3187: L P[3187] 800cm/min CNT100 COORD PTH ;
:SR[23]=$SCR_GRP[1].$MCH_POS_X;
:SR[24]=$SCR_GRP[1].$MCH_POS_Y;
3188: L P[3188] 800cm/min CNT100 COORD PTH ;
:SR[23]=$SCR_GRP[1].$MCH_POS_X;
:SR[24]=$SCR_GRP[1].$MCH_POS_Y;
3189: L P[3189] 800cm/min CNT100 COORD PTH ;
:SR[23]=$SCR_GRP[1].$MCH_POS_X;
:SR[24]=$SCR_GRP[1].$MCH_POS_Y;
3190: L P[3190] 800cm/min CNT100 COORD PTH ;
:SR[23]=$SCR_GRP[1].$MCH_POS_X;
:SR[24]=$SCR_GRP[1].$MCH_POS_Y;
3191: L P[3191] 800cm/min CNT100 COORD PTH ;
:SR[23]=$SCR_GRP[1].$MCH_POS_X;
:SR[24]=$SCR_GRP[1].$MCH_POS_Y;
3192: L P[3192] 800cm/min CNT100 COORD PTH ;
:SR[23]=$SCR_GRP[1].$MCH_POS_X;
:SR[24]=$SCR_GRP[1].$MCH_POS_Y;
3193: L P[3193] 800cm/min CNT100 COORD PTH ;
:SR[23]=$SCR_GRP[1].$MCH_POS_X;
:SR[24]=$SCR_GRP[1].$MCH_POS_Y;
3194: L P[3194] 800cm/min CNT100 COORD PTH ;
:SR[23]=$SCR_GRP[1].$MCH_POS_X;
:SR[24]=$SCR_GRP[1].$MCH_POS_Y;
3195: L P[3195] 800cm/min CNT100 COORD PTH ;
:SR[23]=$SCR_GRP[1].$MCH_POS_X;
:SR[24]=$SCR_GRP[1].$MCH_POS_Y;
3196: L P[3196] 800cm/min CNT100 COORD PTH ;
:SR[23]=$SCR_GRP[1].$MCH_POS_X;
:SR[24]=$SCR_GRP[1].$MCH_POS_Y;
3197: L P[3197] 800cm/min CNT100 COORD PTH ;
:SR[23]=$SCR_GRP[1].$MCH_POS_X;
:SR[24]=$SCR_GRP[1].$MCH_POS_Y;
3198: L P[3198] 800cm/min CNT100 COORD PTH ;
:SR[23]=$SCR_GRP[1].$MCH_POS_X;
:SR[24]=$SCR_GRP[1].$MCH_POS_Y;
3199: L P[3199] 800cm/min CNT100 COORD PTH ;
:SR[23]=$SCR_GRP[1].$MCH_POS_X;
:SR[24]=$SCR_GRP[1].$MCH_POS_Y;
3200: L P[3200] 800cm/min CNT100 COORD PTH ;
:SR[23]=$SCR_GRP[1].$MCH_POS_X;
:SR[24]=$SCR_GRP[1].$MCH_POS_Y;
3201: L P[3201] 800cm/min CNT100 COORD PTH ;
:SR[23]=$SCR_GRP[1].$MCH_POS_X;
:SR[24]=$SCR_GRP[1].$MCH_POS_Y;
3202: L P[3202] 800cm/min CNT100 COORD PTH ;
:SR[23]=$SCR_GRP[1].$MCH_POS_X;
:SR[24]=$SCR_GRP[1].$MCH_POS_Y;
3203: L P[3203] 800cm/min CNT100 COORD PTH ;
:SR[23]=$SCR_GRP[1].$MCH_POS_X;
:SR[24]=$SCR_GRP[1].$MCH_POS_Y;
3204: L P[3204] 800cm/min CNT100 COORD PTH ;
:SR[23]=$SCR_GRP[1].$MCH_POS_X;
:SR[24]=$SCR_GRP[1].$MCH_POS_Y;
3205: L P[3205] 800cm/min CNT100 COORD PTH ;
:SR[23]=$SCR_GRP[1].$MCH_POS_X;
:SR[24]=$SCR_GRP[1].$MCH_POS_Y;
3206: L P[3206] 800cm/min CNT100 COORD PTH ;
:SR[23]=$SCR_GRP[1].$MCH_POS_X;
:SR[24]=$SCR_GRP[1].$MCH_POS_Y;
3207: L P[3207] 800cm/min CNT100 COORD PTH ;
:SR[23]=$SCR_GRP[1].$MCH_POS_X;
:SR[24]=$SCR_GRP[1].$MCH_POS_Y;
3208: L P[3208] 800cm/min CNT100 COORD PTH ;
:SR[23]=$SCR_GRP[1].$MCH_POS_X;
:SR[24]=$SCR_GRP[1].$MCH_POS_Y;
3209: L P[3209] 800cm/min CNT100 COORD PTH ;
:SR[23]=$SCR_GRP[1].$MCH_POS_X;
:SR[24]=$SCR_GRP[1].$MCH_POS_Y;
3210: L P[3210] 800cm/min CNT100 COORD PTH ;
:SR[23]=$SCR_GRP[1].$MCH_POS_X;
:SR[24]=$SCR_GRP[1].$MCH_POS_Y;
3211: L P[3211] 800cm/min CNT100 COORD PTH ;
:SR[23]=$SCR_GRP[1].$MCH_POS_X;
:SR[24]=$SCR_GRP[1].$MCH_POS_Y;
3212: L P[3212] 800cm/min CNT100 COORD PTH ;
:SR[23]=$SCR_GRP[1].$MCH_POS_X;
:SR[24]=$SCR_GRP[1].$MCH_POS_Y;
3213: L P[3213] 800cm/min CNT100 COORD PTH ;
:SR[23]=$SCR_GRP[1].$MCH_POS_X;
:SR[24]=$SCR_GRP[1].$MCH_POS_Y;
3214: L P[3214] 800cm/min CNT100 COORD PTH ;
:SR[23]=$SCR_GRP[1].$MCH_POS_X;
:SR[24]=$SCR_GRP[1].$MCH_POS_Y;
3215: L P[3215] 800cm/min CNT100 COORD PTH ;
:SR[23]=$SCR_GRP[1].$MCH_POS_X;
:SR[24]=$SCR_GRP[1].$MCH_POS_Y;
3216: L P[3216] 800cm/min CNT100 COORD PTH ;
:SR[23]=$SCR_GRP[1].$MCH_POS_X;
:SR[24]=$SCR_GRP[1].$MCH_POS_Y;
3217: L P[3217] 800cm/min CNT100 COORD PTH ;
:SR[23]=$SCR_GRP[1].$MCH_POS_X;
:SR[24]=$SCR_GRP[1].$MCH_POS_Y;
3218: L P[3218] 800cm/min CNT100 COORD PTH ;
:SR[23]=$SCR_GRP[1].$MCH_POS_X;
:SR[24]=$SCR_GRP[1].$MCH_POS_Y;
3219: L P[3219] 800cm/min CNT100 COORD PTH ;
:SR[23]=$SCR_GRP[1].$MCH_POS_X;
:SR[24]=$SCR_GRP[1].$MCH_POS_Y;
3220: L P[3220] 800cm/min CNT100 COORD PTH ;
:SR[23]=$SCR_GRP[1].$MCH_POS_X;
:SR[24]=$SCR_GRP[1].$MCH_POS_Y;
3221: L P[3221] 800cm/min CNT100 COORD PTH ;
:SR[23]=$SCR_GRP[1].$MCH_POS_X;
:SR[24]=$SCR_GRP[1].$MCH_POS_Y;
3222: L P[3222] 800cm/min CNT100 COORD PTH ;
:SR[23]=$SCR_GRP[1].$MCH_POS_X;
:SR[24]=$SCR_GRP[1].$MCH_POS_Y;
3223: L P[3223] 800cm/min CNT100 COORD PTH ;
:SR[23]=$SCR_GRP[1].$MCH_POS_X;
:SR[24]=$SCR_GRP[1].$MCH_POS_Y;
3224: L P[3224] 800cm/min CNT100 COORD PTH ;
:SR[23]=$SCR_GRP[1].$MCH_POS_X;
:SR[24]=$SCR_GRP[1].$MCH_POS_Y;
3225: L P[3225] 800cm/min CNT100 COORD PTH ;
:SR[23]=$SCR_GRP[1].$MCH_POS_X;
:SR[24]=$SCR_GRP[1].$MCH_POS_Y;
3226: L P[3226] 800cm/min CNT100 COORD PTH ;
:SR[23]=$SCR_GRP[1].$MCH_POS_X;
:SR[24]=$SCR_GRP[1].$MCH_POS_Y;
3227: L P[3227] 800cm/min CNT100 COORD PTH ;
:SR[23]=$SCR_GRP[1].$MCH_POS_X;
:SR[24]=$SCR_GRP[1].$MCH_POS_Y;
3228: L P[3228] 800cm/min CNT100 COORD PTH ;
:SR[23]=$SCR_GRP[1].$MCH_POS_X;
:SR[24]=$SCR_GRP[1].$MCH_POS_Y;
3229: L P[3229] 800cm/min CNT100 COORD PTH ;
:SR[23]=$SCR_GRP[1].$MCH_POS_X;
:SR[24]=$SCR_GRP[1].$MCH_POS_Y;
3230: L P[3230] 800cm/min CNT100 COORD PTH ;
:SR[23]=$SCR_GRP[1].$MCH_POS_X;
:SR[24]=$SCR_GRP[1].$MCH_POS_Y;
3231: L P[3231] 800cm/min CNT100 COORD PTH ;
:SR[23]=$SCR_GRP[1].$MCH_POS_X;
:SR[24]=$SCR_GRP[1].$MCH_POS_Y;
3232: L P[3232] 800cm/min CNT100 COORD PTH ;
:SR[23]=$SCR_GRP[1].$MCH_POS_X;
:SR[24]=$SCR_GRP[1].$MCH_POS_Y;
3233: L P[3233] 800cm/min CNT100 COORD PTH ;
:SR[23]=$SCR_GRP[1].$MCH_POS_X;
:SR[24]=$SCR_GRP[1].$MCH_POS_Y;
3234: L P[3234] 800cm/min CNT100 COORD PTH ;
:SR[23]=$SCR_GRP[1].$MCH_POS_X;
:SR[24]=$SCR_GRP[1].$MCH_POS_Y;
3235: L P[3235] 800cm/min CNT100 COORD PTH ;
:SR[23]=$SCR_GRP[1].$MCH_POS_X;
:SR[24]=$SCR_GRP[1].$MCH_POS_Y;
3236: L P[3236] 800cm/min CNT100 COORD PTH ;
:SR[23]=$SCR_GRP[1].$MCH_POS_X;
:SR[24]=$SCR_GRP[1].$MCH_POS_Y;
3237: L P[3237] 800cm/min CNT100 COORD PTH ;
:SR[23]=$SCR_GRP[1].$MCH_POS_X;
:SR[24]=$SCR_GRP[1].$MCH_POS_Y;
3238: L P[3238] 800cm/min CNT100 COORD PTH ;
:SR[23]=$SCR_GRP[1].$MCH_POS_X;
:SR[24]=$SCR_GRP[1].$MCH_POS_Y;
3239: L P[3239] 800cm/min CNT100 COORD PTH ;
:SR[23]=$SCR_GRP[1].$MCH_POS_X;
:SR[24]=$SCR_GRP[1].$MCH_POS_Y;
3240: L P[3240] 800cm/min CNT100 COORD PTH ;
:SR[23]=$SCR_GRP[1].$MCH_POS_X;
:SR[24]=$SCR_GRP[1].$MCH_POS_Y;
3241: L P[3241] 800cm/min CNT100 COORD PTH ;
:SR[23]=$SCR_GRP[1].$MCH_POS_X;
:SR[24]=$SCR_GRP[1].$MCH_POS_Y;
3242: L P[3242] 800cm/min CNT100 COORD PTH ;
:SR[23]=$SCR_GRP[1].$MCH_POS_X;
:SR[24]=$SCR_GRP[1].$MCH_POS_Y;
3243: L P[3243] 800cm/min CNT100 COORD PTH ;
:SR[23]=$SCR_GRP[1].$MCH_POS_X;
:SR[24]=$SCR_GRP[1].$MCH_POS_Y;
3244: L P[3244] 800cm/min CNT100 COORD PTH ;
:SR[23]=$SCR_GRP[1].$MCH_POS_X;
:SR[24]=$SCR_GRP[1].$MCH_POS_Y;
3245: L P[3245] 800cm/min CNT100 COORD PTH ;
:SR[23]=$SCR_GRP[1].$MCH_POS_X;
:SR[24]=$SCR_GRP[1].$MCH_POS_Y;
3246: L P[3246] 800cm/min CNT100 COORD PTH ;
:SR[23]=$SCR_GRP[1].$MCH_POS_X;
:SR[24]=$SCR_GRP[1].$MCH_POS_Y;
3247: L P[3247] 800cm/min CNT100 COORD PTH ;
:SR[23]=$SCR_GRP[1].$MCH_POS_X;
:SR[24]=$SCR_GRP[1].$MCH_POS_Y;
3248: L P[3248] 800cm/min CNT100 COORD PTH ;
:SR[23]=$SCR_GRP[1].$MCH_POS_X;
:SR[24]=$SCR_GRP[1].$MCH_POS_Y;
3249: L P[3249] 800cm/min CNT100 COORD PTH ;
:SR[23]=$SCR_GRP[1].$MCH_POS_X;
:SR[24]=$SCR_GRP[1].$MCH_POS_Y;
3250: L P[3250] 800cm/min CNT100 COORD PTH ;
:SR[23]=$SCR_GRP[1].$MCH_POS_X;
:SR[24]=$SCR_GRP[1].$MCH_POS_Y;
3251: L P[3251] 800cm/min CNT100 COORD PTH ;
:SR[23]=$SCR_GRP[1].$MCH_POS_X;
:SR[24]=$SCR_GRP[1].$MCH_POS_Y;
3252: L P[3252] 800cm/min CNT100 COORD PTH ;
:SR[23]=$SCR_GRP[1].$MCH_POS_X;
:SR[24]=$SCR_GRP[1].$MCH_POS_Y;
3253: L P[3253] 800cm/min CNT100 COORD PTH ;
:SR[23]=$SCR_GRP[1].$MCH_POS_X;
:SR[24]=$SCR_GRP[1].$MCH_POS_Y;
3254: L P[3254] 800cm/min CNT100 COORD PTH ;
:SR[23]=$SCR_GRP[1].$MCH_POS_X;
:SR[24]=$SCR_GRP[1].$MCH_POS_Y;
3255: L P[3255] 800cm/min CNT100 COORD PTH ;
:SR[23]=$SCR_GRP[1].$MCH_POS_X;
:SR[24]=$SCR_GRP[1].$MCH_POS_Y;
3256: L P[3256] 800cm/min CNT100 COORD PTH ;
:SR[23]=$SCR_GRP[1].$MCH_POS_X;
:SR[24]=$SCR_GRP[1].$MCH_POS_Y;
3257: L P[3257] 800cm/min CNT100 COORD PTH ;
:SR[23]=$SCR_GRP[1].$MCH_POS_X;
:SR[24]=$SCR_GRP[1].$MCH_POS_Y;
3258: L P[3258] 800cm/min CNT100 COORD PTH ;
:SR[23]=$SCR_GRP[1].$MCH_POS_X;
:SR[24]=$SCR_GRP[1].$MCH_POS_Y;
3259: L P[3259] 800cm/min CNT100 COORD PTH ;
:SR[23]=$SCR_GRP[1].$MCH_POS_X;
:SR[24]=$SCR_GRP[1].$MCH_POS_Y;
3260: L P[3260] 800cm/min CNT100 COORD PTH ;
:SR[23]=$SCR_GRP[1].$MCH_POS_X;
:SR[24]=$SCR_GRP[1].$MCH_POS_Y;
3261: L P[3261] 800cm/min CNT100 COORD PTH ;
:SR[23]=$SCR_GRP[1].$MCH_POS_X;
:SR[24]=$SCR_GRP[1].$MCH_POS_Y;
3262: L P[3262] 800cm/min CNT100 COORD PTH ;
:SR[23]=$SCR_GRP[1].$MCH_POS_X;
:SR[24]=$SCR_GRP[1].$MCH_POS_Y;
3263: L P[3263] 800cm/min CNT100 COORD PTH ;
:SR[23]=$SCR_GRP[1].$MCH_POS_X;
:SR[24]=$SCR_GRP[1].$MCH_POS_Y;
3264: L P[3264] 800cm/min CNT100 COORD PTH ;
:SR[23]=$SCR_GRP[1].$MCH_POS_X;
:SR[24]=$SCR_GRP[1].$MCH_POS_Y;
3265: L P[3265] 800cm/min CNT100 COORD PTH ;
:SR[23]=$SCR_GRP[1].$MCH_POS_X;
:SR[24]=$SCR_GRP[1].$MCH_POS_Y;
3266: L P[3266] 800cm/min CNT100 COORD PTH ;
:SR[23]=$SCR_GRP[1].$MCH_POS_X;
:SR[24]=$SCR_GRP[1].$MCH_POS_Y;
3267: L P[3267] 800cm/min CNT100 COORD PTH ;
:SR[23]=$SCR_GRP[1].$MCH_POS_X;
:SR[24]=$SCR_GRP[1].$MCH_POS_Y;
3268: L P[3268] 800cm/min CNT100 COORD PTH ;
:SR[23]=$SCR_GRP[1].$MCH_POS_X;
:SR[24]=$SCR_GRP[1].$MCH_POS_Y;
3269: L P[3269] 800cm/min CNT100 COORD PTH ;
:SR[23]=$SCR_GRP[1].$MCH_POS_X;
:SR[24]=$SCR_GRP[1].$MCH_POS_Y;
3270: L P[3270] 800cm/min CNT100 COORD PTH ;
:SR[23]=$SCR_GRP[1].$MCH_POS_X;
:SR[24]=$SCR_GRP[1].$MCH_POS_Y;
3271: L P[3271] 800cm/min CNT100 COORD PTH ;
:SR[23]=$SCR_GRP[1].$MCH_POS_X;
:SR[24]=$SCR_GRP[1].$MCH_POS_Y;
3272: L P[3272] 800cm/min CNT100 COORD PTH ;
:SR[23]=$SCR_GRP[1].$MCH_POS_X;
:SR[24]=$SCR_GRP[1].$MCH_POS_Y;
3273: L P[3273] 800cm/min CNT100 COORD PTH ;
:SR[23]=$SCR_GRP[1].$MCH_POS_X;
:SR[24]=$SCR_GRP[1].$MCH_POS_Y;
3274: L P[3274] 800cm/min CNT100 COORD PTH ;
:SR[23]=$SCR_GRP[1].$MCH_POS_X;
:SR[24]=$SCR_GRP[1].$MCH_POS_Y;
3275: L P[3275] 800cm/min CNT100 COORD PTH ;
:SR[23]=$SCR_GRP[1].$MCH_POS_X;
:SR[24]=$SCR_GRP[1].$MCH_POS_Y;
3276: L P[3276] 800cm/min CNT100 COORD ;
:SR[23]=$SCR_GRP[1].$MCH_POS_X;
:SR[24]=$SCR_GRP[1].$MCH_POS_Y;
3277: L P[3277] 800cm/min CNT100 COORD PTH ;
:SR[23]=$SCR_GRP[1].$MCH_POS_X;
:SR[24]=$SCR_GRP[1].$MCH_POS_Y;
3278: L P[3278] 800cm/min CNT100 COORD PTH ;
:SR[23]=$SCR_GRP[1].$MCH_POS_X;
:SR[24]=$SCR_GRP[1].$MCH_POS_Y;
3279: L P[3279] 800cm/min CNT100 COORD PTH ;
:SR[23]=$SCR_GRP[1].$MCH_POS_X;
:SR[24]=$SCR_GRP[1].$MCH_POS_Y;
3280: L P[3280] 800cm/min CNT100 COORD PTH ;
:SR[23]=$SCR_GRP[1].$MCH_POS_X;
:SR[24]=$SCR_GRP[1].$MCH_POS_Y;
3281: L P[3281] 800cm/min CNT100 COORD PTH ;
:SR[23]=$SCR_GRP[1].$MCH_POS_X;
:SR[24]=$SCR_GRP[1].$MCH_POS_Y;
3282: L P[3282] 800cm/min CNT100 COORD PTH ;
:SR[23]=$SCR_GRP[1].$MCH_POS_X;
:SR[24]=$SCR_GRP[1].$MCH_POS_Y;
3283: L P[3283] 800cm/min CNT100 COORD PTH ;
:SR[23]=$SCR_GRP[1].$MCH_POS_X;
:SR[24]=$SCR_GRP[1].$MCH_POS_Y;
3284: L P[3284] 800cm/min CNT100 COORD PTH ;
:SR[23]=$SCR_GRP[1].$MCH_POS_X;
:SR[24]=$SCR_GRP[1].$MCH_POS_Y;
3285: L P[3285] 800cm/min CNT100 COORD PTH ;
:SR[23]=$SCR_GRP[1].$MCH_POS_X;
:SR[24]=$SCR_GRP[1].$MCH_POS_Y;
3286: L P[3286] 800cm/min CNT100 COORD PTH ;
:SR[23]=$SCR_GRP[1].$MCH_POS_X;
:SR[24]=$SCR_GRP[1].$MCH_POS_Y;
3287: L P[3287] 800cm/min CNT100 COORD PTH ;
:SR[23]=$SCR_GRP[1].$MCH_POS_X;
:SR[24]=$SCR_GRP[1].$MCH_POS_Y;
3288: L P[3288] 800cm/min CNT100 COORD PTH ;
:SR[23]=$SCR_GRP[1].$MCH_POS_X;
:SR[24]=$SCR_GRP[1].$MCH_POS_Y;
3289: L P[3289] 800cm/min CNT100 COORD PTH ;
:SR[23]=$SCR_GRP[1].$MCH_POS_X;
:SR[24]=$SCR_GRP[1].$MCH_POS_Y;
3290: L P[3290] 800cm/min CNT100 COORD PTH ;
:SR[23]=$SCR_GRP[1].$MCH_POS_X;
:SR[24]=$SCR_GRP[1].$MCH_POS_Y;
3291: L P[3291] 800cm/min CNT100 COORD PTH ;
:SR[23]=$SCR_GRP[1].$MCH_POS_X;
:SR[24]=$SCR_GRP[1].$MCH_POS_Y;
3292: L P[3292] 800cm/min CNT100 COORD PTH ;
:SR[23]=$SCR_GRP[1].$MCH_POS_X;
:SR[24]=$SCR_GRP[1].$MCH_POS_Y;
3293: L P[3293] 800cm/min CNT100 COORD PTH ;
:SR[23]=$SCR_GRP[1].$MCH_POS_X;
:SR[24]=$SCR_GRP[1].$MCH_POS_Y;
3294: L P[3294] 800cm/min CNT100 COORD PTH ;
:SR[23]=$SCR_GRP[1].$MCH_POS_X;
:SR[24]=$SCR_GRP[1].$MCH_POS_Y;
3295: L P[3295] 800cm/min CNT100 COORD PTH ;
:SR[23]=$SCR_GRP[1].$MCH_POS_X;
:SR[24]=$SCR_GRP[1].$MCH_POS_Y;
3296: L P[3296] 800cm/min CNT100 COORD PTH ;
:SR[23]=$SCR_GRP[1].$MCH_POS_X;
:SR[24]=$SCR_GRP[1].$MCH_POS_Y;
3297: L P[3297] 800cm/min CNT100 COORD PTH ;
:SR[23]=$SCR_GRP[1].$MCH_POS_X;
:SR[24]=$SCR_GRP[1].$MCH_POS_Y;
3298: L P[3298] 800cm/min CNT100 COORD PTH ;
:SR[23]=$SCR_GRP[1].$MCH_POS_X;
:SR[24]=$SCR_GRP[1].$MCH_POS_Y;
3299: L P[3299] 800cm/min CNT100 COORD PTH ;
:SR[23]=$SCR_GRP[1].$MCH_POS_X;
:SR[24]=$SCR_GRP[1].$MCH_POS_Y;
3300: L P[3300] 800cm/min CNT100 COORD PTH ;
:SR[23]=$SCR_GRP[1].$MCH_POS_X;
:SR[24]=$SCR_GRP[1].$MCH_POS_Y;
3301: L P[3301] 800cm/min CNT100 COORD PTH ;
:SR[23]=$SCR_GRP[1].$MCH_POS_X;
:SR[24]=$SCR_GRP[1].$MCH_POS_Y;
3302: L P[3302] 800cm/min CNT100 COORD PTH ;
:SR[23]=$SCR_GRP[1].$MCH_POS_X;
:SR[24]=$SCR_GRP[1].$MCH_POS_Y;
3303: L P[3303] 800cm/min CNT100 COORD PTH ;
:SR[23]=$SCR_GRP[1].$MCH_POS_X;
:SR[24]=$SCR_GRP[1].$MCH_POS_Y;
3304: L P[3304] 800cm/min CNT100 COORD PTH ;
:SR[23]=$SCR_GRP[1].$MCH_POS_X;
:SR[24]=$SCR_GRP[1].$MCH_POS_Y;
3305: L P[3305] 800cm/min CNT100 COORD PTH ;
:SR[23]=$SCR_GRP[1].$MCH_POS_X;
:SR[24]=$SCR_GRP[1].$MCH_POS_Y;
3306: L P[3306] 800cm/min CNT100 COORD PTH ;
:SR[23]=$SCR_GRP[1].$MCH_POS_X;
:SR[24]=$SCR_GRP[1].$MCH_POS_Y;
3307: L P[3307] 800cm/min CNT100 COORD PTH ;
:SR[23]=$SCR_GRP[1].$MCH_POS_X;
:SR[24]=$SCR_GRP[1].$MCH_POS_Y;
3308: L P[3308] 800cm/min CNT100 COORD PTH ;
:SR[23]=$SCR_GRP[1].$MCH_POS_X;
:SR[24]=$SCR_GRP[1].$MCH_POS_Y;
3309: L P[3309] 800cm/min CNT100 COORD PTH ;
:SR[23]=$SCR_GRP[1].$MCH_POS_X;
:SR[24]=$SCR_GRP[1].$MCH_POS_Y;
3310: L P[3310] 800cm/min CNT100 COORD PTH ;
:SR[23]=$SCR_GRP[1].$MCH_POS_X;
:SR[24]=$SCR_GRP[1].$MCH_POS_Y;
3311: L P[3311] 800cm/min CNT100 COORD PTH ;
:SR[23]=$SCR_GRP[1].$MCH_POS_X;
:SR[24]=$SCR_GRP[1].$MCH_POS_Y;
3312: L P[3312] 800cm/min CNT100 COORD PTH ;
:SR[23]=$SCR_GRP[1].$MCH_POS_X;
:SR[24]=$SCR_GRP[1].$MCH_POS_Y;
3313: L P[3313] 800cm/min CNT100 COORD PTH ;
:SR[23]=$SCR_GRP[1].$MCH_POS_X;
:SR[24]=$SCR_GRP[1].$MCH_POS_Y;
3314: L P[3314] 800cm/min CNT100 COORD PTH ;
:SR[23]=$SCR_GRP[1].$MCH_POS_X;
:SR[24]=$SCR_GRP[1].$MCH_POS_Y;
3315: L P[3315] 800cm/min CNT100 COORD PTH ;
:SR[23]=$SCR_GRP[1].$MCH_POS_X;
:SR[24]=$SCR_GRP[1].$MCH_POS_Y;
3316: L P[3316] 800cm/min CNT100 COORD PTH ;
:SR[23]=$SCR_GRP[1].$MCH_POS_X;
:SR[24]=$SCR_GRP[1].$MCH_POS_Y;
3317: L P[3317] 800cm/min CNT100 COORD PTH ;
:SR[23]=$SCR_GRP[1].$MCH_POS_X;
:SR[24]=$SCR_GRP[1].$MCH_POS_Y;
3318: L P[3318] 800cm/min CNT100 COORD PTH ;
:SR[23]=$SCR_GRP[1].$MCH_POS_X;
:SR[24]=$SCR_GRP[1].$MCH_POS_Y;
3319: L P[3319] 800cm/min CNT100 COORD PTH ;
:SR[23]=$SCR_GRP[1].$MCH_POS_X;
:SR[24]=$SCR_GRP[1].$MCH_POS_Y;
3320: L P[3320] 800cm/min CNT100 COORD PTH ;
:SR[23]=$SCR_GRP[1].$MCH_POS_X;
:SR[24]=$SCR_GRP[1].$MCH_POS_Y;
3321: L P[3321] 800cm/min CNT100 COORD PTH ;
:SR[23]=$SCR_GRP[1].$MCH_POS_X;
:SR[24]=$SCR_GRP[1].$MCH_POS_Y;
3322: L P[3322] 800cm/min CNT100 COORD PTH ;
:SR[23]=$SCR_GRP[1].$MCH_POS_X;
:SR[24]=$SCR_GRP[1].$MCH_POS_Y;
3323: L P[3323] 800cm/min CNT100 COORD PTH ;
:SR[23]=$SCR_GRP[1].$MCH_POS_X;
:SR[24]=$SCR_GRP[1].$MCH_POS_Y;
3324: L P[3324] 800cm/min CNT100 COORD PTH ;
:SR[23]=$SCR_GRP[1].$MCH_POS_X;
:SR[24]=$SCR_GRP[1].$MCH_POS_Y;
3325: L P[3325] 800cm/min CNT100 COORD PTH ;
:SR[23]=$SCR_GRP[1].$MCH_POS_X;
:SR[24]=$SCR_GRP[1].$MCH_POS_Y;
3326: L P[3326] 800cm/min CNT100 COORD PTH ;
:SR[23]=$SCR_GRP[1].$MCH_POS_X;
:SR[24]=$SCR_GRP[1].$MCH_POS_Y;
3327: L P[3327] 800cm/min CNT100 COORD PTH ;
:SR[23]=$SCR_GRP[1].$MCH_POS_X;
:SR[24]=$SCR_GRP[1].$MCH_POS_Y;
3328: L P[3328] 800cm/min CNT100 COORD PTH ;
:SR[23]=$SCR_GRP[1].$MCH_POS_X;
:SR[24]=$SCR_GRP[1].$MCH_POS_Y;
3329: L P[3329] 800cm/min CNT100 COORD PTH ;
:SR[23]=$SCR_GRP[1].$MCH_POS_X;
:SR[24]=$SCR_GRP[1].$MCH_POS_Y;
3330: L P[3330] 800cm/min CNT100 COORD PTH ;
:SR[23]=$SCR_GRP[1].$MCH_POS_X;
:SR[24]=$SCR_GRP[1].$MCH_POS_Y;
3331: L P[3331] 800cm/min CNT100 COORD PTH ;
:SR[23]=$SCR_GRP[1].$MCH_POS_X;
:SR[24]=$SCR_GRP[1].$MCH_POS_Y;
3332: L P[3332] 800cm/min CNT100 COORD PTH ;
:SR[23]=$SCR_GRP[1].$MCH_POS_X;
:SR[24]=$SCR_GRP[1].$MCH_POS_Y;
3333: L P[3333] 800cm/min CNT100 COORD PTH ;
:SR[23]=$SCR_GRP[1].$MCH_POS_X;
:SR[24]=$SCR_GRP[1].$MCH_POS_Y;
3334: L P[3334] 800cm/min CNT100 COORD PTH ;
:SR[23]=$SCR_GRP[1].$MCH_POS_X;
:SR[24]=$SCR_GRP[1].$MCH_POS_Y;
3335: L P[3335] 800cm/min CNT100 COORD PTH ;
:SR[23]=$SCR_GRP[1].$MCH_POS_X;
:SR[24]=$SCR_GRP[1].$MCH_POS_Y;
3336: L P[3336] 800cm/min CNT100 COORD PTH ;
:SR[23]=$SCR_GRP[1].$MCH_POS_X;
:SR[24]=$SCR_GRP[1].$MCH_POS_Y;
3337: L P[3337] 800cm/min CNT100 COORD PTH ;
:SR[23]=$SCR_GRP[1].$MCH_POS_X;
:SR[24]=$SCR_GRP[1].$MCH_POS_Y;
3338: L P[3338] 800cm/min CNT100 COORD PTH ;
:SR[23]=$SCR_GRP[1].$MCH_POS_X;
:SR[24]=$SCR_GRP[1].$MCH_POS_Y;
3339: L P[3339] 800cm/min CNT100 COORD PTH ;
:SR[23]=$SCR_GRP[1].$MCH_POS_X;
:SR[24]=$SCR_GRP[1].$MCH_POS_Y;
3340: L P[3340] 800cm/min CNT100 COORD PTH ;
:SR[23]=$SCR_GRP[1].$MCH_POS_X;
:SR[24]=$SCR_GRP[1].$MCH_POS_Y;
3341: L P[3341] 800cm/min CNT100 COORD PTH ;
:SR[23]=$SCR_GRP[1].$MCH_POS_X;
:SR[24]=$SCR_GRP[1].$MCH_POS_Y;
3342: L P[3342] 800cm/min CNT100 COORD PTH ;
:SR[23]=$SCR_GRP[1].$MCH_POS_X;
:SR[24]=$SCR_GRP[1].$MCH_POS_Y;
3343: L P[3343] 800cm/min CNT100 COORD PTH ;
:SR[23]=$SCR_GRP[1].$MCH_POS_X;
:SR[24]=$SCR_GRP[1].$MCH_POS_Y;
3344: L P[3344] 800cm/min CNT100 COORD PTH ;
:SR[23]=$SCR_GRP[1].$MCH_POS_X;
:SR[24]=$SCR_GRP[1].$MCH_POS_Y;
3345: L P[3345] 800cm/min CNT100 COORD PTH ;
:SR[23]=$SCR_GRP[1].$MCH_POS_X;
:SR[24]=$SCR_GRP[1].$MCH_POS_Y;
3346: L P[3346] 800cm/min CNT100 COORD PTH ;
:SR[23]=$SCR_GRP[1].$MCH_POS_X;
:SR[24]=$SCR_GRP[1].$MCH_POS_Y;
3347: L P[3347] 800cm/min CNT100 COORD PTH ;
:SR[23]=$SCR_GRP[1].$MCH_POS_X;
:SR[24]=$SCR_GRP[1].$MCH_POS_Y;
3348: L P[3348] 800cm/min CNT100 COORD PTH ;
:SR[23]=$SCR_GRP[1].$MCH_POS_X;
:SR[24]=$SCR_GRP[1].$MCH_POS_Y;
3349: L P[3349] 800cm/min CNT100 COORD PTH ;
:SR[23]=$SCR_GRP[1].$MCH_POS_X;
:SR[24]=$SCR_GRP[1].$MCH_POS_Y;
3350: L P[3350] 800cm/min CNT100 COORD PTH ;
:SR[23]=$SCR_GRP[1].$MCH_POS_X;
:SR[24]=$SCR_GRP[1].$MCH_POS_Y;
3351: L P[3351] 800cm/min CNT100 COORD PTH ;
:SR[23]=$SCR_GRP[1].$MCH_POS_X;
:SR[24]=$SCR_GRP[1].$MCH_POS_Y;
3352: L P[3352] 800cm/min CNT100 COORD PTH ;
:SR[23]=$SCR_GRP[1].$MCH_POS_X;
:SR[24]=$SCR_GRP[1].$MCH_POS_Y;
3353: L P[3353] 800cm/min CNT100 COORD PTH ;
:SR[23]=$SCR_GRP[1].$MCH_POS_X;
:SR[24]=$SCR_GRP[1].$MCH_POS_Y;
3354: L P[3354] 800cm/min CNT100 COORD PTH ;
:SR[23]=$SCR_GRP[1].$MCH_POS_X;
:SR[24]=$SCR_GRP[1].$MCH_POS_Y;
3355: L P[3355] 800cm/min CNT100 COORD PTH ;
:SR[23]=$SCR_GRP[1].$MCH_POS_X;
:SR[24]=$SCR_GRP[1].$MCH_POS_Y;
3356: L P[3356] 800cm/min CNT100 COORD PTH ;
:SR[23]=$SCR_GRP[1].$MCH_POS_X;
:SR[24]=$SCR_GRP[1].$MCH_POS_Y;
3357: L P[3357] 800cm/min CNT100 COORD PTH ;
:SR[23]=$SCR_GRP[1].$MCH_POS_X;
:SR[24]=$SCR_GRP[1].$MCH_POS_Y;
3358: L P[3358] 800cm/min CNT100 COORD PTH ;
:SR[23]=$SCR_GRP[1].$MCH_POS_X;
:SR[24]=$SCR_GRP[1].$MCH_POS_Y;
3359: L P[3359] 800cm/min CNT100 COORD PTH ;
:SR[23]=$SCR_GRP[1].$MCH_POS_X;
:SR[24]=$SCR_GRP[1].$MCH_POS_Y;
3360: L P[3360] 800cm/min CNT100 COORD PTH ;
:SR[23]=$SCR_GRP[1].$MCH_POS_X;
:SR[24]=$SCR_GRP[1].$MCH_POS_Y;
3361: L P[3361] 800cm/min CNT100 COORD PTH ;
:SR[23]=$SCR_GRP[1].$MCH_POS_X;
:SR[24]=$SCR_GRP[1].$MCH_POS_Y;
3362: L P[3362] 800cm/min CNT100 COORD PTH ;
:SR[23]=$SCR_GRP[1].$MCH_POS_X;
:SR[24]=$SCR_GRP[1].$MCH_POS_Y;
3363: L P[3363] 800cm/min CNT100 COORD PTH ;
:SR[23]=$SCR_GRP[1].$MCH_POS_X;
:SR[24]=$SCR_GRP[1].$MCH_POS_Y;
3364: L P[3364] 800cm/min CNT100 COORD PTH ;
:SR[23]=$SCR_GRP[1].$MCH_POS_X;
:SR[24]=$SCR_GRP[1].$MCH_POS_Y;
3365: L P[3365] 800cm/min CNT100 COORD PTH ;
:SR[23]=$SCR_GRP[1].$MCH_POS_X;
:SR[24]=$SCR_GRP[1].$MCH_POS_Y;
3366: L P[3366] 800cm/min CNT100 COORD PTH ;
:SR[23]=$SCR_GRP[1].$MCH_POS_X;
:SR[24]=$SCR_GRP[1].$MCH_POS_Y;
3367: L P[3367] 800cm/min CNT100 COORD PTH ;
:SR[23]=$SCR_GRP[1].$MCH_POS_X;
:SR[24]=$SCR_GRP[1].$MCH_POS_Y;
3368: L P[3368] 800cm/min CNT100 COORD PTH ;
:SR[23]=$SCR_GRP[1].$MCH_POS_X;
:SR[24]=$SCR_GRP[1].$MCH_POS_Y;
3369: L P[3369] 800cm/min CNT100 COORD PTH ;
:SR[23]=$SCR_GRP[1].$MCH_POS_X;
:SR[24]=$SCR_GRP[1].$MCH_POS_Y;
3370: L P[3370] 800cm/min CNT100 COORD PTH ;
:SR[23]=$SCR_GRP[1].$MCH_POS_X;
:SR[24]=$SCR_GRP[1].$MCH_POS_Y;
3371: L P[3371] 800cm/min CNT100 COORD PTH ;
:SR[23]=$SCR_GRP[1].$MCH_POS_X;
:SR[24]=$SCR_GRP[1].$MCH_POS_Y;
3372: L P[3372] 800cm/min CNT100 COORD PTH ;
:SR[23]=$SCR_GRP[1].$MCH_POS_X;
:SR[24]=$SCR_GRP[1].$MCH_POS_Y;
3373: L P[3373] 800cm/min CNT100 COORD PTH ;
:SR[23]=$SCR_GRP[1].$MCH_POS_X;
:SR[24]=$SCR_GRP[1].$MCH_POS_Y;
3374: L P[3374] 800cm/min CNT100 COORD PTH ;
:SR[23]=$SCR_GRP[1].$MCH_POS_X;
:SR[24]=$SCR_GRP[1].$MCH_POS_Y;
3375: L P[3375] 800cm/min CNT100 COORD PTH ;
:SR[23]=$SCR_GRP[1].$MCH_POS_X;
:SR[24]=$SCR_GRP[1].$MCH_POS_Y;
3376: L P[3376] 800cm/min CNT100 COORD PTH ;
:SR[23]=$SCR_GRP[1].$MCH_POS_X;
:SR[24]=$SCR_GRP[1].$MCH_POS_Y;
3377: L P[3377] 800cm/min CNT100 COORD PTH ;
:SR[23]=$SCR_GRP[1].$MCH_POS_X;
:SR[24]=$SCR_GRP[1].$MCH_POS_Y;
3378: L P[3378] 800cm/min CNT100 COORD PTH ;
:SR[23]=$SCR_GRP[1].$MCH_POS_X;
:SR[24]=$SCR_GRP[1].$MCH_POS_Y;
3379: L P[3379] 800cm/min CNT100 COORD PTH ;
:SR[23]=$SCR_GRP[1].$MCH_POS_X;
:SR[24]=$SCR_GRP[1].$MCH_POS_Y;
3380: L P[3380] 800cm/min CNT100 COORD PTH ;
:SR[23]=$SCR_GRP[1].$MCH_POS_X;
:SR[24]=$SCR_GRP[1].$MCH_POS_Y;
3381: L P[3381] 800cm/min CNT100 COORD PTH ;
:SR[23]=$SCR_GRP[1].$MCH_POS_X;
:SR[24]=$SCR_GRP[1].$MCH_POS_Y;
3382: L P[3382] 800cm/min CNT100 COORD PTH ;
:SR[23]=$SCR_GRP[1].$MCH_POS_X;
:SR[24]=$SCR_GRP[1].$MCH_POS_Y;
3383: L P[3383] 800cm/min CNT100 COORD PTH ;
:SR[23]=$SCR_GRP[1].$MCH_POS_X;
:SR[24]=$SCR_GRP[1].$MCH_POS_Y;
3384: L P[3384] 800cm/min CNT100 COORD PTH ;
:SR[23]=$SCR_GRP[1].$MCH_POS_X;
:SR[24]=$SCR_GRP[1].$MCH_POS_Y;
3385: L P[3385] 800cm/min CNT100 COORD PTH ;
:SR[23]=$SCR_GRP[1].$MCH_POS_X;
:SR[24]=$SCR_GRP[1].$MCH_POS_Y;
3386: L P[3386] 800cm/min CNT100 COORD PTH ;
:SR[23]=$SCR_GRP[1].$MCH_POS_X;
:SR[24]=$SCR_GRP[1].$MCH_POS_Y;
3387: L P[3387] 800cm/min CNT100 COORD PTH ;
:SR[23]=$SCR_GRP[1].$MCH_POS_X;
:SR[24]=$SCR_GRP[1].$MCH_POS_Y;
3388: L P[3388] 800cm/min CNT100 COORD PTH ;
:SR[23]=$SCR_GRP[1].$MCH_POS_X;
:SR[24]=$SCR_GRP[1].$MCH_POS_Y;
3389: L P[3389] 800cm/min CNT100 COORD PTH ;
:SR[23]=$SCR_GRP[1].$MCH_POS_X;
:SR[24]=$SCR_GRP[1].$MCH_POS_Y;
3390: L P[3390] 800cm/min CNT100 COORD PTH ;
:SR[23]=$SCR_GRP[1].$MCH_POS_X;
:SR[24]=$SCR_GRP[1].$MCH_POS_Y;
3391: L P[3391] 800cm/min CNT100 COORD PTH ;
:SR[23]=$SCR_GRP[1].$MCH_POS_X;
:SR[24]=$SCR_GRP[1].$MCH_POS_Y;
3392: L P[3392] 800cm/min CNT100 COORD PTH ;
:SR[23]=$SCR_GRP[1].$MCH_POS_X;
:SR[24]=$SCR_GRP[1].$MCH_POS_Y;
3393: L P[3393] 800cm/min CNT100 COORD PTH ;
:SR[23]=$SCR_GRP[1].$MCH_POS_X;
:SR[24]=$SCR_GRP[1].$MCH_POS_Y;
3394: L P[3394] 800cm/min CNT100 COORD PTH ;
:SR[23]=$SCR_GRP[1].$MCH_POS_X;
:SR[24]=$SCR_GRP[1].$MCH_POS_Y;
3395: L P[3395] 800cm/min CNT100 COORD PTH ;
:SR[23]=$SCR_GRP[1].$MCH_POS_X;
:SR[24]=$SCR_GRP[1].$MCH_POS_Y;
3396: L P[3396] 800cm/min CNT100 COORD PTH ;
:SR[23]=$SCR_GRP[1].$MCH_POS_X;
:SR[24]=$SCR_GRP[1].$MCH_POS_Y;
3397: L P[3397] 800cm/min CNT100 COORD PTH ;
:SR[23]=$SCR_GRP[1].$MCH_POS_X;
:SR[24]=$SCR_GRP[1].$MCH_POS_Y;
3398: L P[3398] 800cm/min CNT100 COORD PTH ;
:SR[23]=$SCR_GRP[1].$MCH_POS_X;
:SR[24]=$SCR_GRP[1].$MCH_POS_Y;
3399: L P[3399] 800cm/min CNT100 COORD PTH ;
:SR[23]=$SCR_GRP[1].$MCH_POS_X;
:SR[24]=$SCR_GRP[1].$MCH_POS_Y;
3400: L P[3400] 800cm/min CNT100 COORD PTH ;
:SR[23]=$SCR_GRP[1].$MCH_POS_X;
:SR[24]=$SCR_GRP[1].$MCH_POS_Y;
3401: L P[3401] 800cm/min CNT100 COORD PTH ;
:SR[23]=$SCR_GRP[1].$MCH_POS_X;
:SR[24]=$SCR_GRP[1].$MCH_POS_Y;
3402: L P[3402] 800cm/min CNT100 COORD PTH ;
:SR[23]=$SCR_GRP[1].$MCH_POS_X;
:SR[24]=$SCR_GRP[1].$MCH_POS_Y;
3403: L P[3403] 800cm/min CNT100 COORD PTH ;
:SR[23]=$SCR_GRP[1].$MCH_POS_X;
:SR[24]=$SCR_GRP[1].$MCH_POS_Y;
3404: L P[3404] 800cm/min CNT100 COORD PTH ;
:SR[23]=$SCR_GRP[1].$MCH_POS_X;
:SR[24]=$SCR_GRP[1].$MCH_POS_Y;
3405: L P[3405] 800cm/min CNT100 COORD PTH ;
:SR[23]=$SCR_GRP[1].$MCH_POS_X;
:SR[24]=$SCR_GRP[1].$MCH_POS_Y;
3406: L P[3406] 800cm/min CNT100 COORD PTH ;
:SR[23]=$SCR_GRP[1].$MCH_POS_X;
:SR[24]=$SCR_GRP[1].$MCH_POS_Y;
3407: L P[3407] 800cm/min CNT100 COORD PTH ;
:SR[23]=$SCR_GRP[1].$MCH_POS_X;
:SR[24]=$SCR_GRP[1].$MCH_POS_Y;
3408: L P[3408] 800cm/min CNT100 COORD PTH ;
:SR[23]=$SCR_GRP[1].$MCH_POS_X;
:SR[24]=$SCR_GRP[1].$MCH_POS_Y;
3409: L P[3409] 800cm/min CNT100 COORD PTH ;
:SR[23]=$SCR_GRP[1].$MCH_POS_X;
:SR[24]=$SCR_GRP[1].$MCH_POS_Y;
3410: L P[3410] 800cm/min CNT100 COORD PTH ;
:SR[23]=$SCR_GRP[1].$MCH_POS_X;
:SR[24]=$SCR_GRP[1].$MCH_POS_Y;
3411: L P[3411] 800cm/min CNT100 COORD PTH ;
:SR[23]=$SCR_GRP[1].$MCH_POS_X;
:SR[24]=$SCR_GRP[1].$MCH_POS_Y;
3412: L P[3412] 800cm/min CNT100 COORD PTH ;
:SR[23]=$SCR_GRP[1].$MCH_POS_X;
:SR[24]=$SCR_GRP[1].$MCH_POS_Y;
3413: L P[3413] 800cm/min CNT100 COORD PTH ;
:SR[23]=$SCR_GRP[1].$MCH_POS_X;
:SR[24]=$SCR_GRP[1].$MCH_POS_Y;
3414: L P[3414] 800cm/min CNT100 COORD PTH ;
:SR[23]=$SCR_GRP[1].$MCH_POS_X;
:SR[24]=$SCR_GRP[1].$MCH_POS_Y;
3415: L P[3415] 800cm/min CNT100 COORD PTH ;
:SR[23]=$SCR_GRP[1].$MCH_POS_X;
:SR[24]=$SCR_GRP[1].$MCH_POS_Y;
3416: L P[3416] 800cm/min CNT100 COORD PTH ;
:SR[23]=$SCR_GRP[1].$MCH_POS_X;
:SR[24]=$SCR_GRP[1].$MCH_POS_Y;
3417: L P[3417] 800cm/min CNT100 COORD PTH ;
:SR[23]=$SCR_GRP[1].$MCH_POS_X;
:SR[24]=$SCR_GRP[1].$MCH_POS_Y;
3418: L P[3418] 800cm/min CNT100 COORD PTH ;
:SR[23]=$SCR_GRP[1].$MCH_POS_X;
:SR[24]=$SCR_GRP[1].$MCH_POS_Y;
3419: L P[3419] 800cm/min CNT100 COORD PTH ;
:SR[23]=$SCR_GRP[1].$MCH_POS_X;
:SR[24]=$SCR_GRP[1].$MCH_POS_Y;
3420: L P[3420] 800cm/min CNT100 COORD PTH ;
:SR[23]=$SCR_GRP[1].$MCH_POS_X;
:SR[24]=$SCR_GRP[1].$MCH_POS_Y;
3421: L P[3421] 800cm/min CNT100 COORD PTH ;
:SR[23]=$SCR_GRP[1].$MCH_POS_X;
:SR[24]=$SCR_GRP[1].$MCH_POS_Y;
3422: L P[3422] 800cm/min CNT100 COORD PTH ;
:SR[23]=$SCR_GRP[1].$MCH_POS_X;
:SR[24]=$SCR_GRP[1].$MCH_POS_Y;
3423: L P[3423] 800cm/min CNT100 COORD PTH ;
:SR[23]=$SCR_GRP[1].$MCH_POS_X;
:SR[24]=$SCR_GRP[1].$MCH_POS_Y;
3424: L P[3424] 800cm/min CNT100 COORD PTH ;
:SR[23]=$SCR_GRP[1].$MCH_POS_X;
:SR[24]=$SCR_GRP[1].$MCH_POS_Y;
3425: L P[3425] 800cm/min CNT100 COORD PTH ;
:SR[23]=$SCR_GRP[1].$MCH_POS_X;
:SR[24]=$SCR_GRP[1].$MCH_POS_Y;
3426: L P[3426] 800cm/min CNT100 COORD PTH ;
:SR[23]=$SCR_GRP[1].$MCH_POS_X;
:SR[24]=$SCR_GRP[1].$MCH_POS_Y;
3427: L P[3427] 800cm/min CNT100 COORD PTH ;
:SR[23]=$SCR_GRP[1].$MCH_POS_X;
:SR[24]=$SCR_GRP[1].$MCH_POS_Y;
3428: L P[3428] 800cm/min CNT100 COORD PTH ;
:SR[23]=$SCR_GRP[1].$MCH_POS_X;
:SR[24]=$SCR_GRP[1].$MCH_POS_Y;
3429: L P[3429] 800cm/min CNT100 COORD PTH ;
:SR[23]=$SCR_GRP[1].$MCH_POS_X;
:SR[24]=$SCR_GRP[1].$MCH_POS_Y;
3430: L P[3430] 800cm/min CNT100 COORD PTH ;
:SR[23]=$SCR_GRP[1].$MCH_POS_X;
:SR[24]=$SCR_GRP[1].$MCH_POS_Y;
3431: L P[3431] 800cm/min CNT100 COORD PTH ;
:SR[23]=$SCR_GRP[1].$MCH_POS_X;
:SR[24]=$SCR_GRP[1].$MCH_POS_Y;
3432: L P[3432] 800cm/min CNT100 COORD PTH ;
:SR[23]=$SCR_GRP[1].$MCH_POS_X;
:SR[24]=$SCR_GRP[1].$MCH_POS_Y;
3433: L P[3433] 800cm/min CNT100 COORD PTH ;
:SR[23]=$SCR_GRP[1].$MCH_POS_X;
:SR[24]=$SCR_GRP[1].$MCH_POS_Y;
3434: L P[3434] 800cm/min CNT100 COORD PTH ;
:SR[23]=$SCR_GRP[1].$MCH_POS_X;
:SR[24]=$SCR_GRP[1].$MCH_POS_Y;
3435: L P[3435] 800cm/min CNT100 COORD PTH ;
:SR[23]=$SCR_GRP[1].$MCH_POS_X;
:SR[24]=$SCR_GRP[1].$MCH_POS_Y;
3436: L P[3436] 800cm/min CNT100 COORD PTH ;
:SR[23]=$SCR_GRP[1].$MCH_POS_X;
:SR[24]=$SCR_GRP[1].$MCH_POS_Y;
3437: L P[3437] 800cm/min CNT100 COORD PTH ;
:SR[23]=$SCR_GRP[1].$MCH_POS_X;
:SR[24]=$SCR_GRP[1].$MCH_POS_Y;
3438: L P[3438] 800cm/min CNT100 COORD PTH ;
:SR[23]=$SCR_GRP[1].$MCH_POS_X;
:SR[24]=$SCR_GRP[1].$MCH_POS_Y;
3439: L P[3439] 800cm/min CNT100 COORD PTH ;
:SR[23]=$SCR_GRP[1].$MCH_POS_X;
:SR[24]=$SCR_GRP[1].$MCH_POS_Y;
3440: L P[3440] 800cm/min CNT100 COORD PTH ;
:SR[23]=$SCR_GRP[1].$MCH_POS_X;
:SR[24]=$SCR_GRP[1].$MCH_POS_Y;
3441: L P[3441] 800cm/min CNT100 COORD PTH ;
:SR[23]=$SCR_GRP[1].$MCH_POS_X;
:SR[24]=$SCR_GRP[1].$MCH_POS_Y;
3442: L P[3442] 800cm/min CNT100 COORD PTH ;
:SR[23]=$SCR_GRP[1].$MCH_POS_X;
:SR[24]=$SCR_GRP[1].$MCH_POS_Y;
3443: L P[3443] 800cm/min CNT100 COORD PTH ;
:SR[23]=$SCR_GRP[1].$MCH_POS_X;
:SR[24]=$SCR_GRP[1].$MCH_POS_Y;
3444: L P[3444] 800cm/min CNT100 COORD PTH ;
:SR[23]=$SCR_GRP[1].$MCH_POS_X;
:SR[24]=$SCR_GRP[1].$MCH_POS_Y;
3445: L P[3445] 800cm/min CNT100 COORD PTH ;
:SR[23]=$SCR_GRP[1].$MCH_POS_X;
:SR[24]=$SCR_GRP[1].$MCH_POS_Y;
3446: L P[3446] 800cm/min CNT100 COORD PTH ;
:SR[23]=$SCR_GRP[1].$MCH_POS_X;
:SR[24]=$SCR_GRP[1].$MCH_POS_Y;
3447: L P[3447] 800cm/min CNT100 COORD PTH ;
:SR[23]=$SCR_GRP[1].$MCH_POS_X;
:SR[24]=$SCR_GRP[1].$MCH_POS_Y;
3448: L P[3448] 800cm/min CNT100 COORD PTH ;
:SR[23]=$SCR_GRP[1].$MCH_POS_X;
:SR[24]=$SCR_GRP[1].$MCH_POS_Y;
3449: L P[3449] 800cm/min CNT100 COORD PTH ;
:SR[23]=$SCR_GRP[1].$MCH_POS_X;
:SR[24]=$SCR_GRP[1].$MCH_POS_Y;
3450: L P[3450] 800cm/min CNT100 COORD PTH ;
:SR[23]=$SCR_GRP[1].$MCH_POS_X;
:SR[24]=$SCR_GRP[1].$MCH_POS_Y;
3451: L P[3451] 800cm/min CNT100 COORD PTH ;
:SR[23]=$SCR_GRP[1].$MCH_POS_X;
:SR[24]=$SCR_GRP[1].$MCH_POS_Y;
3452: L P[3452] 800cm/min CNT100 COORD PTH ;
:SR[23]=$SCR_GRP[1].$MCH_POS_X;
:SR[24]=$SCR_GRP[1].$MCH_POS_Y;
3453: L P[3453] 800cm/min CNT100 COORD PTH ;
:SR[23]=$SCR_GRP[1].$MCH_POS_X;
:SR[24]=$SCR_GRP[1].$MCH_POS_Y;
3454: L P[3454] 800cm/min CNT100 COORD PTH ;
:SR[23]=$SCR_GRP[1].$MCH_POS_X;
:SR[24]=$SCR_GRP[1].$MCH_POS_Y;
3455: L P[3455] 800cm/min CNT100 COORD PTH ;
:SR[23]=$SCR_GRP[1].$MCH_POS_X;
:SR[24]=$SCR_GRP[1].$MCH_POS_Y;
3456: L P[3456] 800cm/min CNT100 COORD PTH ;
:SR[23]=$SCR_GRP[1].$MCH_POS_X;
:SR[24]=$SCR_GRP[1].$MCH_POS_Y;
3457: L P[3457] 800cm/min CNT100 COORD PTH ;
:SR[23]=$SCR_GRP[1].$MCH_POS_X;
:SR[24]=$SCR_GRP[1].$MCH_POS_Y;
3458: L P[3458] 800cm/min CNT100 COORD PTH ;
:SR[23]=$SCR_GRP[1].$MCH_POS_X;
:SR[24]=$SCR_GRP[1].$MCH_POS_Y;
3459: L P[3459] 800cm/min CNT100 COORD PTH ;
:SR[23]=$SCR_GRP[1].$MCH_POS_X;
:SR[24]=$SCR_GRP[1].$MCH_POS_Y;
3460: L P[3460] 800cm/min CNT100 COORD PTH ;
:SR[23]=$SCR_GRP[1].$MCH_POS_X;
:SR[24]=$SCR_GRP[1].$MCH_POS_Y;
3461: L P[3461] 800cm/min CNT100 COORD PTH ;
:SR[23]=$SCR_GRP[1].$MCH_POS_X;
:SR[24]=$SCR_GRP[1].$MCH_POS_Y;
3462: L P[3462] 800cm/min CNT100 COORD PTH ;
:SR[23]=$SCR_GRP[1].$MCH_POS_X;
:SR[24]=$SCR_GRP[1].$MCH_POS_Y;
3463: L P[3463] 800cm/min CNT100 COORD PTH ;
:SR[23]=$SCR_GRP[1].$MCH_POS_X;
:SR[24]=$SCR_GRP[1].$MCH_POS_Y;
3464: L P[3464] 800cm/min CNT100 COORD PTH ;
:SR[23]=$SCR_GRP[1].$MCH_POS_X;
:SR[24]=$SCR_GRP[1].$MCH_POS_Y;
3465: L P[3465] 800cm/min CNT100 COORD PTH ;
:SR[23]=$SCR_GRP[1].$MCH_POS_X;
:SR[24]=$SCR_GRP[1].$MCH_POS_Y;
3466: L P[3466] 800cm/min CNT100 COORD PTH ;
:SR[23]=$SCR_GRP[1].$MCH_POS_X;
:SR[24]=$SCR_GRP[1].$MCH_POS_Y;
3467: L P[3467] 800cm/min CNT100 COORD PTH ;
:SR[23]=$SCR_GRP[1].$MCH_POS_X;
:SR[24]=$SCR_GRP[1].$MCH_POS_Y;
3468: L P[3468] 800cm/min CNT100 COORD PTH ;
:SR[23]=$SCR_GRP[1].$MCH_POS_X;
:SR[24]=$SCR_GRP[1].$MCH_POS_Y;
3469: L P[3469] 800cm/min CNT100 COORD PTH ;
:SR[23]=$SCR_GRP[1].$MCH_POS_X;
:SR[24]=$SCR_GRP[1].$MCH_POS_Y;
3470: L P[3470] 800cm/min CNT100 COORD PTH ;
:SR[23]=$SCR_GRP[1].$MCH_POS_X;
:SR[24]=$SCR_GRP[1].$MCH_POS_Y;
3471: L P[3471] 800cm/min CNT100 COORD PTH ;
:SR[23]=$SCR_GRP[1].$MCH_POS_X;
:SR[24]=$SCR_GRP[1].$MCH_POS_Y;
3472: L P[3472] 800cm/min CNT100 COORD PTH ;
:SR[23]=$SCR_GRP[1].$MCH_POS_X;
:SR[24]=$SCR_GRP[1].$MCH_POS_Y;
3473: L P[3473] 800cm/min CNT100 COORD PTH ;
:SR[23]=$SCR_GRP[1].$MCH_POS_X;
:SR[24]=$SCR_GRP[1].$MCH_POS_Y;
3474: L P[3474] 800cm/min CNT100 COORD PTH ;
:SR[23]=$SCR_GRP[1].$MCH_POS_X;
:SR[24]=$SCR_GRP[1].$MCH_POS_Y;
3475: L P[3475] 800cm/min CNT100 COORD PTH ;
:SR[23]=$SCR_GRP[1].$MCH_POS_X;
:SR[24]=$SCR_GRP[1].$MCH_POS_Y;
3476: L P[3476] 800cm/min CNT100 COORD PTH ;
:SR[23]=$SCR_GRP[1].$MCH_POS_X;
:SR[24]=$SCR_GRP[1].$MCH_POS_Y;
3477: L P[3477] 800cm/min CNT100 COORD PTH ;
:SR[23]=$SCR_GRP[1].$MCH_POS_X;
:SR[24]=$SCR_GRP[1].$MCH_POS_Y;
3478: L P[3478] 800cm/min CNT100 COORD PTH ;
:SR[23]=$SCR_GRP[1].$MCH_POS_X;
:SR[24]=$SCR_GRP[1].$MCH_POS_Y;
3479: L P[3479] 800cm/min CNT100 COORD PTH ;
:SR[23]=$SCR_GRP[1].$MCH_POS_X;
:SR[24]=$SCR_GRP[1].$MCH_POS_Y;
3480: L P[3480] 800cm/min CNT100 COORD PTH ;
:SR[23]=$SCR_GRP[1].$MCH_POS_X;
:SR[24]=$SCR_GRP[1].$MCH_POS_Y;
3481: L P[3481] 800cm/min CNT100 COORD PTH ;
:SR[23]=$SCR_GRP[1].$MCH_POS_X;
:SR[24]=$SCR_GRP[1].$MCH_POS_Y;
3482: L P[3482] 800cm/min CNT100 COORD PTH ;
:SR[23]=$SCR_GRP[1].$MCH_POS_X;
:SR[24]=$SCR_GRP[1].$MCH_POS_Y;
3483: L P[3483] 800cm/min CNT100 COORD PTH ;
:SR[23]=$SCR_GRP[1].$MCH_POS_X;
:SR[24]=$SCR_GRP[1].$MCH_POS_Y;
3484: L P[3484] 800cm/min CNT100 COORD PTH ;
:SR[23]=$SCR_GRP[1].$MCH_POS_X;
:SR[24]=$SCR_GRP[1].$MCH_POS_Y;
3485: L P[3485] 800cm/min CNT100 COORD PTH ;
:SR[23]=$SCR_GRP[1].$MCH_POS_X;
:SR[24]=$SCR_GRP[1].$MCH_POS_Y;
3486: L P[3486] 800cm/min CNT100 COORD PTH ;
:SR[23]=$SCR_GRP[1].$MCH_POS_X;
:SR[24]=$SCR_GRP[1].$MCH_POS_Y;
3487: L P[3487] 800cm/min CNT100 COORD PTH ;
:SR[23]=$SCR_GRP[1].$MCH_POS_X;
:SR[24]=$SCR_GRP[1].$MCH_POS_Y;
3488: L P[3488] 800cm/min CNT100 COORD PTH ;
:SR[23]=$SCR_GRP[1].$MCH_POS_X;
:SR[24]=$SCR_GRP[1].$MCH_POS_Y;
3489: L P[3489] 800cm/min CNT100 COORD PTH ;
:SR[23]=$SCR_GRP[1].$MCH_POS_X;
:SR[24]=$SCR_GRP[1].$MCH_POS_Y;
3490: L P[3490] 800cm/min CNT100 COORD PTH ;
:SR[23]=$SCR_GRP[1].$MCH_POS_X;
:SR[24]=$SCR_GRP[1].$MCH_POS_Y;
3491: L P[3491] 800cm/min CNT100 COORD PTH ;
:SR[23]=$SCR_GRP[1].$MCH_POS_X;
:SR[24]=$SCR_GRP[1].$MCH_POS_Y;
3492: L P[3492] 800cm/min CNT100 COORD PTH ;
:SR[23]=$SCR_GRP[1].$MCH_POS_X;
:SR[24]=$SCR_GRP[1].$MCH_POS_Y;
3493: L P[3493] 800cm/min CNT100 COORD PTH ;
:SR[23]=$SCR_GRP[1].$MCH_POS_X;
:SR[24]=$SCR_GRP[1].$MCH_POS_Y;
3494: L P[3494] 800cm/min CNT100 COORD PTH ;
:SR[23]=$SCR_GRP[1].$MCH_POS_X;
:SR[24]=$SCR_GRP[1].$MCH_POS_Y;
3495: L P[3495] 800cm/min CNT100 COORD PTH ;
:SR[23]=$SCR_GRP[1].$MCH_POS_X;
:SR[24]=$SCR_GRP[1].$MCH_POS_Y;
3496: L P[3496] 800cm/min CNT100 COORD PTH ;
:SR[23]=$SCR_GRP[1].$MCH_POS_X;
:SR[24]=$SCR_GRP[1].$MCH_POS_Y;
3497: L P[3497] 800cm/min CNT100 COORD PTH ;
:SR[23]=$SCR_GRP[1].$MCH_POS_X;
:SR[24]=$SCR_GRP[1].$MCH_POS_Y;
3498: L P[3498] 800cm/min CNT100 COORD PTH ;
:SR[23]=$SCR_GRP[1].$MCH_POS_X;
:SR[24]=$SCR_GRP[1].$MCH_POS_Y;
3499: L P[3499] 800cm/min CNT100 COORD PTH ;
:SR[23]=$SCR_GRP[1].$MCH_POS_X;
:SR[24]=$SCR_GRP[1].$MCH_POS_Y;
3500: L P[3500] 800cm/min CNT100 COORD PTH ;
:SR[23]=$SCR_GRP[1].$MCH_POS_X;
:SR[24]=$SCR_GRP[1].$MCH_POS_Y;
3501: L P[3501] 800cm/min CNT100 COORD PTH ;
:SR[23]=$SCR_GRP[1].$MCH_POS_X;
:SR[24]=$SCR_GRP[1].$MCH_POS_Y;
3502: L P[3502] 800cm/min CNT100 COORD PTH ;
:SR[23]=$SCR_GRP[1].$MCH_POS_X;
:SR[24]=$SCR_GRP[1].$MCH_POS_Y;
3503: L P[3503] 800cm/min CNT100 COORD PTH ;
:SR[23]=$SCR_GRP[1].$MCH_POS_X;
:SR[24]=$SCR_GRP[1].$MCH_POS_Y;
3504: L P[3504] 800cm/min CNT100 COORD PTH ;
:SR[23]=$SCR_GRP[1].$MCH_POS_X;
:SR[24]=$SCR_GRP[1].$MCH_POS_Y;
3505: L P[3505] 800cm/min CNT100 COORD PTH ;
:SR[23]=$SCR_GRP[1].$MCH_POS_X;
:SR[24]=$SCR_GRP[1].$MCH_POS_Y;
3506: L P[3506] 800cm/min CNT100 COORD PTH ;
:SR[23]=$SCR_GRP[1].$MCH_POS_X;
:SR[24]=$SCR_GRP[1].$MCH_POS_Y;
3507: L P[3507] 800cm/min CNT100 COORD PTH ;
:SR[23]=$SCR_GRP[1].$MCH_POS_X;
:SR[24]=$SCR_GRP[1].$MCH_POS_Y;
3508: L P[3508] 800cm/min CNT100 COORD PTH ;
:SR[23]=$SCR_GRP[1].$MCH_POS_X;
:SR[24]=$SCR_GRP[1].$MCH_POS_Y;
3509: L P[3509] 800cm/min CNT100 COORD PTH ;
:SR[23]=$SCR_GRP[1].$MCH_POS_X;
:SR[24]=$SCR_GRP[1].$MCH_POS_Y;
3510: L P[3510] 800cm/min CNT100 COORD PTH ;
:SR[23]=$SCR_GRP[1].$MCH_POS_X;
:SR[24]=$SCR_GRP[1].$MCH_POS_Y;
3511: L P[3511] 800cm/min CNT100 COORD PTH ;
:SR[23]=$SCR_GRP[1].$MCH_POS_X;
:SR[24]=$SCR_GRP[1].$MCH_POS_Y;
3512: L P[3512] 800cm/min CNT100 COORD PTH ;
:SR[23]=$SCR_GRP[1].$MCH_POS_X;
:SR[24]=$SCR_GRP[1].$MCH_POS_Y;
3513: L P[3513] 800cm/min CNT100 COORD PTH ;
:SR[23]=$SCR_GRP[1].$MCH_POS_X;
:SR[24]=$SCR_GRP[1].$MCH_POS_Y;
3514: L P[3514] 800cm/min CNT100 COORD PTH ;
:SR[23]=$SCR_GRP[1].$MCH_POS_X;
:SR[24]=$SCR_GRP[1].$MCH_POS_Y;
3515: L P[3515] 800cm/min CNT100 COORD PTH ;
:SR[23]=$SCR_GRP[1].$MCH_POS_X;
:SR[24]=$SCR_GRP[1].$MCH_POS_Y;
3516: L P[3516] 800cm/min CNT100 COORD PTH ;
:SR[23]=$SCR_GRP[1].$MCH_POS_X;
:SR[24]=$SCR_GRP[1].$MCH_POS_Y;
3517: L P[3517] 800cm/min CNT100 COORD PTH ;
:SR[23]=$SCR_GRP[1].$MCH_POS_X;
:SR[24]=$SCR_GRP[1].$MCH_POS_Y;
3518: L P[3518] 800cm/min CNT100 COORD PTH ;
:SR[23]=$SCR_GRP[1].$MCH_POS_X;
:SR[24]=$SCR_GRP[1].$MCH_POS_Y;
3519: L P[3519] 800cm/min CNT100 COORD PTH ;
:SR[23]=$SCR_GRP[1].$MCH_POS_X;
:SR[24]=$SCR_GRP[1].$MCH_POS_Y;
3520: L P[3520] 800cm/min CNT100 COORD PTH ;
:SR[23]=$SCR_GRP[1].$MCH_POS_X;
:SR[24]=$SCR_GRP[1].$MCH_POS_Y;
3521: L P[3521] 800cm/min CNT100 COORD PTH ;
:SR[23]=$SCR_GRP[1].$MCH_POS_X;
:SR[24]=$SCR_GRP[1].$MCH_POS_Y;
3522: L P[3522] 800cm/min CNT100 COORD PTH ;
:SR[23]=$SCR_GRP[1].$MCH_POS_X;
:SR[24]=$SCR_GRP[1].$MCH_POS_Y;
3523: L P[3523] 800cm/min CNT100 COORD PTH ;
:SR[23]=$SCR_GRP[1].$MCH_POS_X;
:SR[24]=$SCR_GRP[1].$MCH_POS_Y;
3524: L P[3524] 800cm/min CNT100 COORD PTH ;
:SR[23]=$SCR_GRP[1].$MCH_POS_X;
:SR[24]=$SCR_GRP[1].$MCH_POS_Y;
3525: L P[3525] 800cm/min CNT100 COORD PTH ;
:SR[23]=$SCR_GRP[1].$MCH_POS_X;
:SR[24]=$SCR_GRP[1].$MCH_POS_Y;
3526: L P[3526] 800cm/min CNT100 COORD PTH ;
:SR[23]=$SCR_GRP[1].$MCH_POS_X;
:SR[24]=$SCR_GRP[1].$MCH_POS_Y;
3527: L P[3527] 800cm/min CNT100 COORD PTH ;
:SR[23]=$SCR_GRP[1].$MCH_POS_X;
:SR[24]=$SCR_GRP[1].$MCH_POS_Y;
3528: L P[3528] 800cm/min CNT100 COORD PTH ;
:SR[23]=$SCR_GRP[1].$MCH_POS_X;
:SR[24]=$SCR_GRP[1].$MCH_POS_Y;
3529: L P[3529] 800cm/min CNT100 COORD PTH ;
:SR[23]=$SCR_GRP[1].$MCH_POS_X;
:SR[24]=$SCR_GRP[1].$MCH_POS_Y;
3530: L P[3530] 800cm/min CNT100 COORD PTH ;
:SR[23]=$SCR_GRP[1].$MCH_POS_X;
:SR[24]=$SCR_GRP[1].$MCH_POS_Y;
3531: L P[3531] 800cm/min CNT100 COORD PTH ;
:SR[23]=$SCR_GRP[1].$MCH_POS_X;
:SR[24]=$SCR_GRP[1].$MCH_POS_Y;
3532: L P[3532] 800cm/min CNT100 COORD PTH ;
:SR[23]=$SCR_GRP[1].$MCH_POS_X;
:SR[24]=$SCR_GRP[1].$MCH_POS_Y;
3533: L P[3533] 800cm/min CNT100 COORD PTH ;
:SR[23]=$SCR_GRP[1].$MCH_POS_X;
:SR[24]=$SCR_GRP[1].$MCH_POS_Y;
3534: L P[3534] 800cm/min CNT100 COORD PTH ;
:SR[23]=$SCR_GRP[1].$MCH_POS_X;
:SR[24]=$SCR_GRP[1].$MCH_POS_Y;
3535: L P[3535] 800cm/min CNT100 COORD PTH ;
:SR[23]=$SCR_GRP[1].$MCH_POS_X;
:SR[24]=$SCR_GRP[1].$MCH_POS_Y;
3536: L P[3536] 800cm/min CNT100 COORD PTH ;
:SR[23]=$SCR_GRP[1].$MCH_POS_X;
:SR[24]=$SCR_GRP[1].$MCH_POS_Y;
3537: L P[3537] 800cm/min CNT100 COORD PTH ;
:SR[23]=$SCR_GRP[1].$MCH_POS_X;
:SR[24]=$SCR_GRP[1].$MCH_POS_Y;
3538: L P[3538] 800cm/min CNT100 COORD PTH ;
:SR[23]=$SCR_GRP[1].$MCH_POS_X;
:SR[24]=$SCR_GRP[1].$MCH_POS_Y;
3539: L P[3539] 800cm/min CNT100 COORD PTH ;
:SR[23]=$SCR_GRP[1].$MCH_POS_X;
:SR[24]=$SCR_GRP[1].$MCH_POS_Y;
3540: L P[3540] 800cm/min CNT100 COORD PTH ;
:SR[23]=$SCR_GRP[1].$MCH_POS_X;
:SR[24]=$SCR_GRP[1].$MCH_POS_Y;
3541: L P[3541] 800cm/min CNT100 COORD PTH ;
:SR[23]=$SCR_GRP[1].$MCH_POS_X;
:SR[24]=$SCR_GRP[1].$MCH_POS_Y;
3542: L P[3542] 800cm/min CNT100 COORD PTH ;
:SR[23]=$SCR_GRP[1].$MCH_POS_X;
:SR[24]=$SCR_GRP[1].$MCH_POS_Y;
3543: L P[3543] 800cm/min CNT100 COORD PTH ;
:SR[23]=$SCR_GRP[1].$MCH_POS_X;
:SR[24]=$SCR_GRP[1].$MCH_POS_Y;
3544: L P[3544] 800cm/min CNT100 COORD PTH ;
:SR[23]=$SCR_GRP[1].$MCH_POS_X;
:SR[24]=$SCR_GRP[1].$MCH_POS_Y;
3545: L P[3545] 800cm/min CNT100 COORD PTH ;
:SR[23]=$SCR_GRP[1].$MCH_POS_X;
:SR[24]=$SCR_GRP[1].$MCH_POS_Y;
3546: L P[3546] 800cm/min CNT100 COORD PTH ;
:SR[23]=$SCR_GRP[1].$MCH_POS_X;
:SR[24]=$SCR_GRP[1].$MCH_POS_Y;
3547: L P[3547] 800cm/min CNT100 COORD PTH ;
:SR[23]=$SCR_GRP[1].$MCH_POS_X;
:SR[24]=$SCR_GRP[1].$MCH_POS_Y;
3548: L P[3548] 800cm/min CNT100 COORD PTH ;
:SR[23]=$SCR_GRP[1].$MCH_POS_X;
:SR[24]=$SCR_GRP[1].$MCH_POS_Y;
3549: L P[3549] 800cm/min CNT100 COORD PTH ;
:SR[23]=$SCR_GRP[1].$MCH_POS_X;
:SR[24]=$SCR_GRP[1].$MCH_POS_Y;
3550: L P[3550] 800cm/min CNT100 COORD PTH ;
:SR[23]=$SCR_GRP[1].$MCH_POS_X;
:SR[24]=$SCR_GRP[1].$MCH_POS_Y;
3551: L P[3551] 800cm/min CNT100 COORD PTH ;
:SR[23]=$SCR_GRP[1].$MCH_POS_X;
:SR[24]=$SCR_GRP[1].$MCH_POS_Y;
3552: L P[3552] 800cm/min CNT100 COORD PTH ;
:SR[23]=$SCR_GRP[1].$MCH_POS_X;
:SR[24]=$SCR_GRP[1].$MCH_POS_Y;
3553: L P[3553] 800cm/min CNT100 COORD PTH ;
:SR[23]=$SCR_GRP[1].$MCH_POS_X;
:SR[24]=$SCR_GRP[1].$MCH_POS_Y;
3554: L P[3554] 800cm/min CNT100 COORD PTH ;
:SR[23]=$SCR_GRP[1].$MCH_POS_X;
:SR[24]=$SCR_GRP[1].$MCH_POS_Y;
3555: L P[3555] 800cm/min CNT100 COORD PTH ;
:SR[23]=$SCR_GRP[1].$MCH_POS_X;
:SR[24]=$SCR_GRP[1].$MCH_POS_Y;
3556: L P[3556] 800cm/min CNT100 COORD PTH ;
:SR[23]=$SCR_GRP[1].$MCH_POS_X;
:SR[24]=$SCR_GRP[1].$MCH_POS_Y;
3557: L P[3557] 800cm/min CNT100 COORD PTH ;
:SR[23]=$SCR_GRP[1].$MCH_POS_X;
:SR[24]=$SCR_GRP[1].$MCH_POS_Y;
3558: L P[3558] 800cm/min CNT100 COORD PTH ;
:SR[23]=$SCR_GRP[1].$MCH_POS_X;
:SR[24]=$SCR_GRP[1].$MCH_POS_Y;
3559: L P[3559] 800cm/min CNT100 COORD PTH ;
:SR[23]=$SCR_GRP[1].$MCH_POS_X;
:SR[24]=$SCR_GRP[1].$MCH_POS_Y;
3560: L P[3560] 800cm/min CNT100 COORD PTH ;
:SR[23]=$SCR_GRP[1].$MCH_POS_X;
:SR[24]=$SCR_GRP[1].$MCH_POS_Y;
3561: L P[3561] 800cm/min CNT100 COORD PTH ;
:SR[23]=$SCR_GRP[1].$MCH_POS_X;
:SR[24]=$SCR_GRP[1].$MCH_POS_Y;
3562: L P[3562] 800cm/min CNT100 COORD PTH ;
:SR[23]=$SCR_GRP[1].$MCH_POS_X;
:SR[24]=$SCR_GRP[1].$MCH_POS_Y;
3563: L P[3563] 800cm/min CNT100 COORD PTH ;
:SR[23]=$SCR_GRP[1].$MCH_POS_X;
:SR[24]=$SCR_GRP[1].$MCH_POS_Y;
3564: L P[3564] 800cm/min CNT100 COORD PTH ;
:SR[23]=$SCR_GRP[1].$MCH_POS_X;
:SR[24]=$SCR_GRP[1].$MCH_POS_Y;
3565: L P[3565] 800cm/min CNT100 COORD PTH ;
:SR[23]=$SCR_GRP[1].$MCH_POS_X;
:SR[24]=$SCR_GRP[1].$MCH_POS_Y;
3566: L P[3566] 800cm/min CNT100 COORD PTH ;
:SR[23]=$SCR_GRP[1].$MCH_POS_X;
:SR[24]=$SCR_GRP[1].$MCH_POS_Y;
3567: L P[3567] 800cm/min CNT100 COORD PTH ;
:SR[23]=$SCR_GRP[1].$MCH_POS_X;
:SR[24]=$SCR_GRP[1].$MCH_POS_Y;
3568: L P[3568] 800cm/min CNT100 COORD PTH ;
:SR[23]=$SCR_GRP[1].$MCH_POS_X;
:SR[24]=$SCR_GRP[1].$MCH_POS_Y;
3569: L P[3569] 800cm/min CNT100 COORD PTH ;
:SR[23]=$SCR_GRP[1].$MCH_POS_X;
:SR[24]=$SCR_GRP[1].$MCH_POS_Y;
3570: L P[3570] 800cm/min CNT100 COORD PTH ;
:SR[23]=$SCR_GRP[1].$MCH_POS_X;
:SR[24]=$SCR_GRP[1].$MCH_POS_Y;
3571: L P[3571] 800cm/min CNT100 COORD PTH ;
:SR[23]=$SCR_GRP[1].$MCH_POS_X;
:SR[24]=$SCR_GRP[1].$MCH_POS_Y;
3572: L P[3572] 800cm/min CNT100 COORD PTH ;
:SR[23]=$SCR_GRP[1].$MCH_POS_X;
:SR[24]=$SCR_GRP[1].$MCH_POS_Y;
3573: L P[3573] 800cm/min CNT100 COORD PTH ;
:SR[23]=$SCR_GRP[1].$MCH_POS_X;
:SR[24]=$SCR_GRP[1].$MCH_POS_Y;
3574: L P[3574] 800cm/min CNT100 COORD PTH ;
:SR[23]=$SCR_GRP[1].$MCH_POS_X;
:SR[24]=$SCR_GRP[1].$MCH_POS_Y;
3575: L P[3575] 800cm/min CNT100 COORD PTH ;
:SR[23]=$SCR_GRP[1].$MCH_POS_X;
:SR[24]=$SCR_GRP[1].$MCH_POS_Y;
3576: L P[3576] 800cm/min CNT100 COORD PTH ;
:SR[23]=$SCR_GRP[1].$MCH_POS_X;
:SR[24]=$SCR_GRP[1].$MCH_POS_Y;
3577: L P[3577] 800cm/min CNT100 COORD PTH ;
:SR[23]=$SCR_GRP[1].$MCH_POS_X;
:SR[24]=$SCR_GRP[1].$MCH_POS_Y;
3578: L P[3578] 800cm/min CNT100 COORD PTH ;
:SR[23]=$SCR_GRP[1].$MCH_POS_X;
:SR[24]=$SCR_GRP[1].$MCH_POS_Y;
3579: L P[3579] 800cm/min CNT100 COORD PTH ;
:SR[23]=$SCR_GRP[1].$MCH_POS_X;
:SR[24]=$SCR_GRP[1].$MCH_POS_Y;
3580: L P[3580] 800cm/min CNT100 COORD PTH ;
:SR[23]=$SCR_GRP[1].$MCH_POS_X;
:SR[24]=$SCR_GRP[1].$MCH_POS_Y;
3581: L P[3581] 800cm/min CNT100 COORD PTH ;
:SR[23]=$SCR_GRP[1].$MCH_POS_X;
:SR[24]=$SCR_GRP[1].$MCH_POS_Y;
3582: L P[3582] 800cm/min CNT100 COORD PTH ;
:SR[23]=$SCR_GRP[1].$MCH_POS_X;
:SR[24]=$SCR_GRP[1].$MCH_POS_Y;
3583: L P[3583] 800cm/min CNT100 COORD PTH ;
:SR[23]=$SCR_GRP[1].$MCH_POS_X;
:SR[24]=$SCR_GRP[1].$MCH_POS_Y;
3584: L P[3584] 800cm/min CNT100 COORD PTH ;
:SR[23]=$SCR_GRP[1].$MCH_POS_X;
:SR[24]=$SCR_GRP[1].$MCH_POS_Y;
3585: L P[3585] 800cm/min CNT100 COORD PTH ;
:SR[23]=$SCR_GRP[1].$MCH_POS_X;
:SR[24]=$SCR_GRP[1].$MCH_POS_Y;
3586: L P[3586] 800cm/min CNT100 COORD PTH ;
:SR[23]=$SCR_GRP[1].$MCH_POS_X;
:SR[24]=$SCR_GRP[1].$MCH_POS_Y;
3587: L P[3587] 800cm/min CNT100 COORD PTH ;
:SR[23]=$SCR_GRP[1].$MCH_POS_X;
:SR[24]=$SCR_GRP[1].$MCH_POS_Y;
3588: L P[3588] 800cm/min CNT100 COORD PTH ;
:SR[23]=$SCR_GRP[1].$MCH_POS_X;
:SR[24]=$SCR_GRP[1].$MCH_POS_Y;
3589: L P[3589] 800cm/min CNT100 COORD PTH ;
:SR[23]=$SCR_GRP[1].$MCH_POS_X;
:SR[24]=$SCR_GRP[1].$MCH_POS_Y;
3590: L P[3590] 800cm/min CNT100 COORD PTH ;
:SR[23]=$SCR_GRP[1].$MCH_POS_X;
:SR[24]=$SCR_GRP[1].$MCH_POS_Y;
3591: L P[3591] 800cm/min CNT100 COORD PTH ;
:SR[23]=$SCR_GRP[1].$MCH_POS_X;
:SR[24]=$SCR_GRP[1].$MCH_POS_Y;
3592: L P[3592] 800cm/min CNT100 COORD PTH ;
:SR[23]=$SCR_GRP[1].$MCH_POS_X;
:SR[24]=$SCR_GRP[1].$MCH_POS_Y;
3593: L P[3593] 800cm/min CNT100 COORD PTH ;
:SR[23]=$SCR_GRP[1].$MCH_POS_X;
:SR[24]=$SCR_GRP[1].$MCH_POS_Y;
3594: L P[3594] 800cm/min CNT100 COORD PTH ;
:SR[23]=$SCR_GRP[1].$MCH_POS_X;
:SR[24]=$SCR_GRP[1].$MCH_POS_Y;
3595: L P[3595] 800cm/min CNT100 COORD PTH ;
:SR[23]=$SCR_GRP[1].$MCH_POS_X;
:SR[24]=$SCR_GRP[1].$MCH_POS_Y;
3596: L P[3596] 800cm/min CNT100 COORD PTH ;
:SR[23]=$SCR_GRP[1].$MCH_POS_X;
:SR[24]=$SCR_GRP[1].$MCH_POS_Y;
3597: L P[3597] 800cm/min CNT100 COORD PTH ;
:SR[23]=$SCR_GRP[1].$MCH_POS_X;
:SR[24]=$SCR_GRP[1].$MCH_POS_Y;
3598: L P[3598] 800cm/min CNT100 COORD PTH ;
:SR[23]=$SCR_GRP[1].$MCH_POS_X;
:SR[24]=$SCR_GRP[1].$MCH_POS_Y;
3599: L P[3599] 800cm/min CNT100 COORD PTH ;
:SR[23]=$SCR_GRP[1].$MCH_POS_X;
:SR[24]=$SCR_GRP[1].$MCH_POS_Y;
3600: L P[3600] 800cm/min CNT100 COORD PTH ;
:SR[23]=$SCR_GRP[1].$MCH_POS_X;
:SR[24]=$SCR_GRP[1].$MCH_POS_Y;
3601: L P[3601] 800cm/min CNT100 COORD PTH ;
:SR[23]=$SCR_GRP[1].$MCH_POS_X;
:SR[24]=$SCR_GRP[1].$MCH_POS_Y;
3602: L P[3602] 800cm/min CNT100 COORD PTH ;
:SR[23]=$SCR_GRP[1].$MCH_POS_X;
:SR[24]=$SCR_GRP[1].$MCH_POS_Y;
3603: L P[3603] 800cm/min CNT100 COORD PTH ;
:SR[23]=$SCR_GRP[1].$MCH_POS_X;
:SR[24]=$SCR_GRP[1].$MCH_POS_Y;
3604: L P[3604] 800cm/min CNT100 COORD PTH ;
:SR[23]=$SCR_GRP[1].$MCH_POS_X;
:SR[24]=$SCR_GRP[1].$MCH_POS_Y;
3605: L P[3605] 800cm/min CNT100 COORD PTH ;
:SR[23]=$SCR_GRP[1].$MCH_POS_X;
:SR[24]=$SCR_GRP[1].$MCH_POS_Y;
3606: L P[3606] 800cm/min CNT100 COORD PTH ;
:SR[23]=$SCR_GRP[1].$MCH_POS_X;
:SR[24]=$SCR_GRP[1].$MCH_POS_Y;
3607: L P[3607] 800cm/min CNT100 COORD PTH ;
:SR[23]=$SCR_GRP[1].$MCH_POS_X;
:SR[24]=$SCR_GRP[1].$MCH_POS_Y;
3608: L P[3608] 800cm/min CNT100 COORD PTH ;
:SR[23]=$SCR_GRP[1].$MCH_POS_X;
:SR[24]=$SCR_GRP[1].$MCH_POS_Y;
3609: L P[3609] 800cm/min CNT100 COORD PTH ;
:SR[23]=$SCR_GRP[1].$MCH_POS_X;
:SR[24]=$SCR_GRP[1].$MCH_POS_Y;
3610: L P[3610] 800cm/min CNT100 COORD PTH ;
:SR[23]=$SCR_GRP[1].$MCH_POS_X;
:SR[24]=$SCR_GRP[1].$MCH_POS_Y;
3611: L P[3611] 800cm/min CNT100 COORD PTH ;
:SR[23]=$SCR_GRP[1].$MCH_POS_X;
:SR[24]=$SCR_GRP[1].$MCH_POS_Y;
3612: L P[3612] 800cm/min CNT100 COORD PTH ;
:SR[23]=$SCR_GRP[1].$MCH_POS_X;
:SR[24]=$SCR_GRP[1].$MCH_POS_Y;
3613: L P[3613] 800cm/min CNT100 COORD PTH ;
:SR[23]=$SCR_GRP[1].$MCH_POS_X;
:SR[24]=$SCR_GRP[1].$MCH_POS_Y;
3614: L P[3614] 800cm/min CNT100 COORD PTH ;
:SR[23]=$SCR_GRP[1].$MCH_POS_X;
:SR[24]=$SCR_GRP[1].$MCH_POS_Y;
3615: L P[3615] 800cm/min CNT100 COORD PTH ;
:SR[23]=$SCR_GRP[1].$MCH_POS_X;
:SR[24]=$SCR_GRP[1].$MCH_POS_Y;
3616: L P[3616] 800cm/min CNT100 COORD PTH ;
:SR[23]=$SCR_GRP[1].$MCH_POS_X;
:SR[24]=$SCR_GRP[1].$MCH_POS_Y;
3617: L P[3617] 800cm/min CNT100 COORD PTH ;
:SR[23]=$SCR_GRP[1].$MCH_POS_X;
:SR[24]=$SCR_GRP[1].$MCH_POS_Y;
3618: L P[3618] 800cm/min CNT100 COORD PTH ;
:SR[23]=$SCR_GRP[1].$MCH_POS_X;
:SR[24]=$SCR_GRP[1].$MCH_POS_Y;
3619: L P[3619] 800cm/min CNT100 COORD PTH ;
:SR[23]=$SCR_GRP[1].$MCH_POS_X;
:SR[24]=$SCR_GRP[1].$MCH_POS_Y;
3620: L P[3620] 800cm/min CNT100 COORD PTH ;
:SR[23]=$SCR_GRP[1].$MCH_POS_X;
:SR[24]=$SCR_GRP[1].$MCH_POS_Y;
3621: L P[3621] 800cm/min CNT100 COORD PTH ;
:SR[23]=$SCR_GRP[1].$MCH_POS_X;
:SR[24]=$SCR_GRP[1].$MCH_POS_Y;
3622: L P[3622] 800cm/min CNT100 COORD PTH ;
:SR[23]=$SCR_GRP[1].$MCH_POS_X;
:SR[24]=$SCR_GRP[1].$MCH_POS_Y;
3623: L P[3623] 800cm/min CNT100 COORD PTH ;
:SR[23]=$SCR_GRP[1].$MCH_POS_X;
:SR[24]=$SCR_GRP[1].$MCH_POS_Y;
3624: L P[3624] 800cm/min CNT100 COORD PTH ;
:SR[23]=$SCR_GRP[1].$MCH_POS_X;
:SR[24]=$SCR_GRP[1].$MCH_POS_Y;
3625: L P[3625] 800cm/min CNT100 COORD PTH ;
:SR[23]=$SCR_GRP[1].$MCH_POS_X;
:SR[24]=$SCR_GRP[1].$MCH_POS_Y;
3626: L P[3626] 800cm/min CNT100 COORD PTH ;
:SR[23]=$SCR_GRP[1].$MCH_POS_X;
:SR[24]=$SCR_GRP[1].$MCH_POS_Y;
3627: L P[3627] 800cm/min CNT100 COORD PTH ;
:SR[23]=$SCR_GRP[1].$MCH_POS_X;
:SR[24]=$SCR_GRP[1].$MCH_POS_Y;
3628: L P[3628] 800cm/min CNT100 COORD PTH ;
:SR[23]=$SCR_GRP[1].$MCH_POS_X;
:SR[24]=$SCR_GRP[1].$MCH_POS_Y;
3629: L P[3629] 800cm/min CNT100 COORD PTH ;
:SR[23]=$SCR_GRP[1].$MCH_POS_X;
:SR[24]=$SCR_GRP[1].$MCH_POS_Y;
3630: L P[3630] 800cm/min CNT100 COORD PTH ;
:SR[23]=$SCR_GRP[1].$MCH_POS_X;
:SR[24]=$SCR_GRP[1].$MCH_POS_Y;
3631: L P[3631] 800cm/min CNT100 COORD PTH ;
:SR[23]=$SCR_GRP[1].$MCH_POS_X;
:SR[24]=$SCR_GRP[1].$MCH_POS_Y;
3632: L P[3632] 800cm/min CNT100 COORD PTH ;
:SR[23]=$SCR_GRP[1].$MCH_POS_X;
:SR[24]=$SCR_GRP[1].$MCH_POS_Y;
3633: L P[3633] 800cm/min CNT100 COORD PTH ;
:SR[23]=$SCR_GRP[1].$MCH_POS_X;
:SR[24]=$SCR_GRP[1].$MCH_POS_Y;
3634: L P[3634] 800cm/min CNT100 COORD PTH ;
:SR[23]=$SCR_GRP[1].$MCH_POS_X;
:SR[24]=$SCR_GRP[1].$MCH_POS_Y;
3635: L P[3635] 800cm/min CNT100 COORD PTH ;
:SR[23]=$SCR_GRP[1].$MCH_POS_X;
:SR[24]=$SCR_GRP[1].$MCH_POS_Y;
3636: L P[3636] 800cm/min CNT100 COORD PTH ;
:SR[23]=$SCR_GRP[1].$MCH_POS_X;
:SR[24]=$SCR_GRP[1].$MCH_POS_Y;
3637: L P[3637] 800cm/min CNT100 COORD PTH ;
:SR[23]=$SCR_GRP[1].$MCH_POS_X;
:SR[24]=$SCR_GRP[1].$MCH_POS_Y;
3638: L P[3638] 800cm/min CNT100 COORD PTH ;
:SR[23]=$SCR_GRP[1].$MCH_POS_X;
:SR[24]=$SCR_GRP[1].$MCH_POS_Y;
3639: L P[3639] 800cm/min CNT100 COORD PTH ;
:SR[23]=$SCR_GRP[1].$MCH_POS_X;
:SR[24]=$SCR_GRP[1].$MCH_POS_Y;
3640: L P[3640] 800cm/min CNT100 COORD PTH ;
:SR[23]=$SCR_GRP[1].$MCH_POS_X;
:SR[24]=$SCR_GRP[1].$MCH_POS_Y;
3641: L P[3641] 800cm/min CNT100 COORD PTH ;
:SR[23]=$SCR_GRP[1].$MCH_POS_X;
:SR[24]=$SCR_GRP[1].$MCH_POS_Y;
3642: L P[3642] 800cm/min CNT100 COORD PTH ;
:SR[23]=$SCR_GRP[1].$MCH_POS_X;
:SR[24]=$SCR_GRP[1].$MCH_POS_Y;
3643: L P[3643] 800cm/min CNT100 COORD PTH ;
:SR[23]=$SCR_GRP[1].$MCH_POS_X;
:SR[24]=$SCR_GRP[1].$MCH_POS_Y;
3644: L P[3644] 800cm/min CNT100 COORD PTH ;
:SR[23]=$SCR_GRP[1].$MCH_POS_X;
:SR[24]=$SCR_GRP[1].$MCH_POS_Y;
3645: L P[3645] 800cm/min CNT100 COORD PTH ;
:SR[23]=$SCR_GRP[1].$MCH_POS_X;
:SR[24]=$SCR_GRP[1].$MCH_POS_Y;
3646: L P[3646] 800cm/min CNT100 COORD PTH ;
:SR[23]=$SCR_GRP[1].$MCH_POS_X;
:SR[24]=$SCR_GRP[1].$MCH_POS_Y;
3647: L P[3647] 800cm/min CNT100 COORD PTH ;
:SR[23]=$SCR_GRP[1].$MCH_POS_X;
:SR[24]=$SCR_GRP[1].$MCH_POS_Y;
3648: L P[3648] 800cm/min CNT100 COORD PTH ;
:SR[23]=$SCR_GRP[1].$MCH_POS_X;
:SR[24]=$SCR_GRP[1].$MCH_POS_Y;
3649: L P[3649] 800cm/min CNT100 COORD PTH ;
:SR[23]=$SCR_GRP[1].$MCH_POS_X;
:SR[24]=$SCR_GRP[1].$MCH_POS_Y;
3650: L P[3650] 800cm/min CNT100 COORD PTH ;
:SR[23]=$SCR_GRP[1].$MCH_POS_X;
:SR[24]=$SCR_GRP[1].$MCH_POS_Y;
3651: L P[3651] 800cm/min CNT100 COORD PTH ;
:SR[23]=$SCR_GRP[1].$MCH_POS_X;
:SR[24]=$SCR_GRP[1].$MCH_POS_Y;
3652: L P[3652] 800cm/min CNT100 COORD PTH ;
:SR[23]=$SCR_GRP[1].$MCH_POS_X;
:SR[24]=$SCR_GRP[1].$MCH_POS_Y;
3653: L P[3653] 800cm/min CNT100 COORD PTH ;
:SR[23]=$SCR_GRP[1].$MCH_POS_X;
:SR[24]=$SCR_GRP[1].$MCH_POS_Y;
3654: L P[3654] 800cm/min CNT100 COORD PTH ;
:SR[23]=$SCR_GRP[1].$MCH_POS_X;
:SR[24]=$SCR_GRP[1].$MCH_POS_Y;
3655: L P[3655] 800cm/min CNT100 COORD PTH ;
:SR[23]=$SCR_GRP[1].$MCH_POS_X;
:SR[24]=$SCR_GRP[1].$MCH_POS_Y;
3656: L P[3656] 800cm/min CNT100 COORD PTH ;
:SR[23]=$SCR_GRP[1].$MCH_POS_X;
:SR[24]=$SCR_GRP[1].$MCH_POS_Y;
3657: L P[3657] 800cm/min CNT100 COORD PTH ;
:SR[23]=$SCR_GRP[1].$MCH_POS_X;
:SR[24]=$SCR_GRP[1].$MCH_POS_Y;
3658: L P[3658] 800cm/min CNT100 COORD PTH ;
:SR[23]=$SCR_GRP[1].$MCH_POS_X;
:SR[24]=$SCR_GRP[1].$MCH_POS_Y;
3659: L P[3659] 800cm/min CNT100 COORD PTH ;
:SR[23]=$SCR_GRP[1].$MCH_POS_X;
:SR[24]=$SCR_GRP[1].$MCH_POS_Y;
3660: L P[3660] 800cm/min CNT100 COORD PTH ;
:SR[23]=$SCR_GRP[1].$MCH_POS_X;
:SR[24]=$SCR_GRP[1].$MCH_POS_Y;
3661: L P[3661] 800cm/min CNT100 COORD PTH ;
:SR[23]=$SCR_GRP[1].$MCH_POS_X;
:SR[24]=$SCR_GRP[1].$MCH_POS_Y;
3662: L P[3662] 800cm/min CNT100 COORD PTH ;
:SR[23]=$SCR_GRP[1].$MCH_POS_X;
:SR[24]=$SCR_GRP[1].$MCH_POS_Y;
3663: L P[3663] 800cm/min CNT100 COORD PTH ;
:SR[23]=$SCR_GRP[1].$MCH_POS_X;
:SR[24]=$SCR_GRP[1].$MCH_POS_Y;
3664: L P[3664] 800cm/min CNT100 COORD PTH ;
:SR[23]=$SCR_GRP[1].$MCH_POS_X;
:SR[24]=$SCR_GRP[1].$MCH_POS_Y;
3665: L P[3665] 800cm/min CNT100 COORD PTH ;
:SR[23]=$SCR_GRP[1].$MCH_POS_X;
:SR[24]=$SCR_GRP[1].$MCH_POS_Y;
3666: L P[3666] 800cm/min CNT100 COORD PTH ;
:SR[23]=$SCR_GRP[1].$MCH_POS_X;
:SR[24]=$SCR_GRP[1].$MCH_POS_Y;
3667: L P[3667] 800cm/min CNT100 COORD PTH ;
:SR[23]=$SCR_GRP[1].$MCH_POS_X;
:SR[24]=$SCR_GRP[1].$MCH_POS_Y;
3668: L P[3668] 800cm/min CNT100 COORD PTH ;
:SR[23]=$SCR_GRP[1].$MCH_POS_X;
:SR[24]=$SCR_GRP[1].$MCH_POS_Y;
3669: L P[3669] 800cm/min CNT100 COORD PTH ;
:SR[23]=$SCR_GRP[1].$MCH_POS_X;
:SR[24]=$SCR_GRP[1].$MCH_POS_Y;
3670: L P[3670] 800cm/min CNT100 COORD PTH ;
:SR[23]=$SCR_GRP[1].$MCH_POS_X;
:SR[24]=$SCR_GRP[1].$MCH_POS_Y;
3671: L P[3671] 800cm/min CNT100 COORD PTH ;
:SR[23]=$SCR_GRP[1].$MCH_POS_X;
:SR[24]=$SCR_GRP[1].$MCH_POS_Y;
3672: L P[3672] 800cm/min CNT100 COORD PTH ;
:SR[23]=$SCR_GRP[1].$MCH_POS_X;
:SR[24]=$SCR_GRP[1].$MCH_POS_Y;
3673: L P[3673] 800cm/min CNT100 COORD PTH ;
:SR[23]=$SCR_GRP[1].$MCH_POS_X;
:SR[24]=$SCR_GRP[1].$MCH_POS_Y;
3674: L P[3674] 800cm/min CNT100 COORD PTH ;
:SR[23]=$SCR_GRP[1].$MCH_POS_X;
:SR[24]=$SCR_GRP[1].$MCH_POS_Y;
3675: L P[3675] 800cm/min CNT100 COORD PTH ;
:SR[23]=$SCR_GRP[1].$MCH_POS_X;
:SR[24]=$SCR_GRP[1].$MCH_POS_Y;
3676: L P[3676] 800cm/min CNT100 COORD PTH ;
:SR[23]=$SCR_GRP[1].$MCH_POS_X;
:SR[24]=$SCR_GRP[1].$MCH_POS_Y;
3677: L P[3677] 800cm/min CNT100 COORD PTH ;
:SR[23]=$SCR_GRP[1].$MCH_POS_X;
:SR[24]=$SCR_GRP[1].$MCH_POS_Y;
3678: L P[3678] 800cm/min CNT100 COORD PTH ;
:SR[23]=$SCR_GRP[1].$MCH_POS_X;
:SR[24]=$SCR_GRP[1].$MCH_POS_Y;
3679: L P[3679] 800cm/min CNT100 COORD PTH ;
:SR[23]=$SCR_GRP[1].$MCH_POS_X;
:SR[24]=$SCR_GRP[1].$MCH_POS_Y;
3680: L P[3680] 800cm/min CNT100 COORD PTH ;
:SR[23]=$SCR_GRP[1].$MCH_POS_X;
:SR[24]=$SCR_GRP[1].$MCH_POS_Y;
3681: L P[3681] 800cm/min CNT100 COORD PTH ;
:SR[23]=$SCR_GRP[1].$MCH_POS_X;
:SR[24]=$SCR_GRP[1].$MCH_POS_Y;
3682: L P[3682] 800cm/min CNT100 COORD PTH ;
:SR[23]=$SCR_GRP[1].$MCH_POS_X;
:SR[24]=$SCR_GRP[1].$MCH_POS_Y;
3683: L P[3683] 800cm/min CNT100 COORD PTH ;
:SR[23]=$SCR_GRP[1].$MCH_POS_X;
:SR[24]=$SCR_GRP[1].$MCH_POS_Y;
3684: L P[3684] 800cm/min CNT100 COORD PTH ;
:SR[23]=$SCR_GRP[1].$MCH_POS_X;
:SR[24]=$SCR_GRP[1].$MCH_POS_Y;
3685: L P[3685] 800cm/min CNT100 COORD PTH ;
:SR[23]=$SCR_GRP[1].$MCH_POS_X;
:SR[24]=$SCR_GRP[1].$MCH_POS_Y;
3686: L P[3686] 800cm/min CNT100 COORD PTH ;
:SR[23]=$SCR_GRP[1].$MCH_POS_X;
:SR[24]=$SCR_GRP[1].$MCH_POS_Y;
3687: L P[3687] 800cm/min CNT100 COORD PTH ;
:SR[23]=$SCR_GRP[1].$MCH_POS_X;
:SR[24]=$SCR_GRP[1].$MCH_POS_Y;
3688: L P[3688] 800cm/min CNT100 COORD PTH ;
:SR[23]=$SCR_GRP[1].$MCH_POS_X;
:SR[24]=$SCR_GRP[1].$MCH_POS_Y;
3689: L P[3689] 800cm/min CNT100 COORD PTH ;
:SR[23]=$SCR_GRP[1].$MCH_POS_X;
:SR[24]=$SCR_GRP[1].$MCH_POS_Y;
3690: L P[3690] 800cm/min CNT100 COORD PTH ;
:SR[23]=$SCR_GRP[1].$MCH_POS_X;
:SR[24]=$SCR_GRP[1].$MCH_POS_Y;
3691: L P[3691] 800cm/min CNT100 COORD PTH ;
:SR[23]=$SCR_GRP[1].$MCH_POS_X;
:SR[24]=$SCR_GRP[1].$MCH_POS_Y;
3692: L P[3692] 800cm/min CNT100 COORD PTH ;
:SR[23]=$SCR_GRP[1].$MCH_POS_X;
:SR[24]=$SCR_GRP[1].$MCH_POS_Y;
3693: L P[3693] 800cm/min CNT100 COORD PTH ;
:SR[23]=$SCR_GRP[1].$MCH_POS_X;
:SR[24]=$SCR_GRP[1].$MCH_POS_Y;
3694: L P[3694] 800cm/min CNT100 COORD PTH ;
:SR[23]=$SCR_GRP[1].$MCH_POS_X;
:SR[24]=$SCR_GRP[1].$MCH_POS_Y;
3695: L P[3695] 800cm/min CNT100 COORD PTH ;
:SR[23]=$SCR_GRP[1].$MCH_POS_X;
:SR[24]=$SCR_GRP[1].$MCH_POS_Y;
3696: L P[3696] 800cm/min CNT100 COORD PTH ;
:SR[23]=$SCR_GRP[1].$MCH_POS_X;
:SR[24]=$SCR_GRP[1].$MCH_POS_Y;
3697: L P[3697] 800cm/min CNT100 COORD PTH ;
:SR[23]=$SCR_GRP[1].$MCH_POS_X;
:SR[24]=$SCR_GRP[1].$MCH_POS_Y;
3698: L P[3698] 800cm/min CNT100 COORD PTH ;
:SR[23]=$SCR_GRP[1].$MCH_POS_X;
:SR[24]=$SCR_GRP[1].$MCH_POS_Y;
3699: L P[3699] 800cm/min CNT100 COORD PTH ;
:SR[23]=$SCR_GRP[1].$MCH_POS_X;
:SR[24]=$SCR_GRP[1].$MCH_POS_Y;
3700: L P[3700] 800cm/min CNT100 COORD PTH ;
:SR[23]=$SCR_GRP[1].$MCH_POS_X;
:SR[24]=$SCR_GRP[1].$MCH_POS_Y;
3701: L P[3701] 800cm/min CNT100 COORD PTH ;
:SR[23]=$SCR_GRP[1].$MCH_POS_X;
:SR[24]=$SCR_GRP[1].$MCH_POS_Y;
3702: L P[3702] 800cm/min CNT100 COORD PTH ;
:SR[23]=$SCR_GRP[1].$MCH_POS_X;
:SR[24]=$SCR_GRP[1].$MCH_POS_Y;
3703: L P[3703] 800cm/min CNT100 COORD PTH ;
:SR[23]=$SCR_GRP[1].$MCH_POS_X;
:SR[24]=$SCR_GRP[1].$MCH_POS_Y;
3704: L P[3704] 800cm/min CNT100 COORD PTH ;
:SR[23]=$SCR_GRP[1].$MCH_POS_X;
:SR[24]=$SCR_GRP[1].$MCH_POS_Y;
3705: L P[3705] 800cm/min CNT100 COORD PTH ;
:SR[23]=$SCR_GRP[1].$MCH_POS_X;
:SR[24]=$SCR_GRP[1].$MCH_POS_Y;
3706: L P[3706] 800cm/min CNT100 COORD PTH ;
:SR[23]=$SCR_GRP[1].$MCH_POS_X;
:SR[24]=$SCR_GRP[1].$MCH_POS_Y;
3707: L P[3707] 800cm/min CNT100 COORD PTH ;
:SR[23]=$SCR_GRP[1].$MCH_POS_X;
:SR[24]=$SCR_GRP[1].$MCH_POS_Y;
3708: L P[3708] 800cm/min CNT100 COORD PTH ;
:SR[23]=$SCR_GRP[1].$MCH_POS_X;
:SR[24]=$SCR_GRP[1].$MCH_POS_Y;
3709: L P[3709] 800cm/min CNT100 COORD PTH ;
:SR[23]=$SCR_GRP[1].$MCH_POS_X;
:SR[24]=$SCR_GRP[1].$MCH_POS_Y;
3710: L P[3710] 800cm/min CNT100 COORD PTH ;
:SR[23]=$SCR_GRP[1].$MCH_POS_X;
:SR[24]=$SCR_GRP[1].$MCH_POS_Y;
3711: L P[3711] 800cm/min CNT100 COORD PTH ;
:SR[23]=$SCR_GRP[1].$MCH_POS_X;
:SR[24]=$SCR_GRP[1].$MCH_POS_Y;
3712: L P[3712] 800cm/min CNT100 COORD PTH ;
:SR[23]=$SCR_GRP[1].$MCH_POS_X;
:SR[24]=$SCR_GRP[1].$MCH_POS_Y;
3713: L P[3713] 800cm/min CNT100 COORD PTH ;
:SR[23]=$SCR_GRP[1].$MCH_POS_X;
:SR[24]=$SCR_GRP[1].$MCH_POS_Y;
3714: L P[3714] 800cm/min CNT100 COORD PTH ;
:SR[23]=$SCR_GRP[1].$MCH_POS_X;
:SR[24]=$SCR_GRP[1].$MCH_POS_Y;
3715: L P[3715] 800cm/min CNT100 COORD PTH ;
:SR[23]=$SCR_GRP[1].$MCH_POS_X;
:SR[24]=$SCR_GRP[1].$MCH_POS_Y;
3716: L P[3716] 800cm/min CNT100 COORD PTH ;
:SR[23]=$SCR_GRP[1].$MCH_POS_X;
:SR[24]=$SCR_GRP[1].$MCH_POS_Y;
3717: L P[3717] 800cm/min CNT100 COORD PTH ;
:SR[23]=$SCR_GRP[1].$MCH_POS_X;
:SR[24]=$SCR_GRP[1].$MCH_POS_Y;
3718: L P[3718] 800cm/min CNT100 COORD PTH ;
:SR[23]=$SCR_GRP[1].$MCH_POS_X;
:SR[24]=$SCR_GRP[1].$MCH_POS_Y;
3719: L P[3719] 800cm/min CNT100 COORD PTH ;
:SR[23]=$SCR_GRP[1].$MCH_POS_X;
:SR[24]=$SCR_GRP[1].$MCH_POS_Y;
3720: L P[3720] 800cm/min CNT100 COORD PTH ;
:SR[23]=$SCR_GRP[1].$MCH_POS_X;
:SR[24]=$SCR_GRP[1].$MCH_POS_Y;
3721: L P[3721] 800cm/min CNT100 COORD PTH ;
:SR[23]=$SCR_GRP[1].$MCH_POS_X;
:SR[24]=$SCR_GRP[1].$MCH_POS_Y;
3722: L P[3722] 800cm/min CNT100 COORD PTH ;
:SR[23]=$SCR_GRP[1].$MCH_POS_X;
:SR[24]=$SCR_GRP[1].$MCH_POS_Y;
3723: L P[3723] 800cm/min CNT100 COORD PTH ;
:SR[23]=$SCR_GRP[1].$MCH_POS_X;
:SR[24]=$SCR_GRP[1].$MCH_POS_Y;
3724: L P[3724] 800cm/min CNT100 COORD PTH ;
:SR[23]=$SCR_GRP[1].$MCH_POS_X;
:SR[24]=$SCR_GRP[1].$MCH_POS_Y;
3725: L P[3725] 800cm/min CNT100 COORD PTH ;
:SR[23]=$SCR_GRP[1].$MCH_POS_X;
:SR[24]=$SCR_GRP[1].$MCH_POS_Y;
3726: L P[3726] 800cm/min CNT100 COORD PTH ;
:SR[23]=$SCR_GRP[1].$MCH_POS_X;
:SR[24]=$SCR_GRP[1].$MCH_POS_Y;
3727: L P[3727] 800cm/min CNT100 COORD PTH ;
:SR[23]=$SCR_GRP[1].$MCH_POS_X;
:SR[24]=$SCR_GRP[1].$MCH_POS_Y;
3728: L P[3728] 800cm/min CNT100 COORD PTH ;
:SR[23]=$SCR_GRP[1].$MCH_POS_X;
:SR[24]=$SCR_GRP[1].$MCH_POS_Y;
3729: L P[3729] 800cm/min CNT100 COORD PTH ;
:SR[23]=$SCR_GRP[1].$MCH_POS_X;
:SR[24]=$SCR_GRP[1].$MCH_POS_Y;
3730: L P[3730] 800cm/min CNT100 COORD PTH ;
:SR[23]=$SCR_GRP[1].$MCH_POS_X;
:SR[24]=$SCR_GRP[1].$MCH_POS_Y;
3731: L P[3731] 800cm/min CNT100 COORD PTH ;
:SR[23]=$SCR_GRP[1].$MCH_POS_X;
:SR[24]=$SCR_GRP[1].$MCH_POS_Y;
3732: L P[3732] 800cm/min CNT100 COORD PTH ;
:SR[23]=$SCR_GRP[1].$MCH_POS_X;
:SR[24]=$SCR_GRP[1].$MCH_POS_Y;
3733: L P[3733] 800cm/min CNT100 COORD PTH ;
:SR[23]=$SCR_GRP[1].$MCH_POS_X;
:SR[24]=$SCR_GRP[1].$MCH_POS_Y;
3734: L P[3734] 800cm/min CNT100 COORD PTH ;
:SR[23]=$SCR_GRP[1].$MCH_POS_X;
:SR[24]=$SCR_GRP[1].$MCH_POS_Y;
3735: L P[3735] 800cm/min CNT100 COORD PTH ;
:SR[23]=$SCR_GRP[1].$MCH_POS_X;
:SR[24]=$SCR_GRP[1].$MCH_POS_Y;
3736: L P[3736] 800cm/min CNT100 COORD PTH ;
:SR[23]=$SCR_GRP[1].$MCH_POS_X;
:SR[24]=$SCR_GRP[1].$MCH_POS_Y;
3737: L P[3737] 800cm/min CNT100 COORD PTH ;
:SR[23]=$SCR_GRP[1].$MCH_POS_X;
:SR[24]=$SCR_GRP[1].$MCH_POS_Y;
3738: L P[3738] 800cm/min CNT100 COORD PTH ;
:SR[23]=$SCR_GRP[1].$MCH_POS_X;
:SR[24]=$SCR_GRP[1].$MCH_POS_Y;
3739: L P[3739] 800cm/min CNT100 COORD PTH ;
:SR[23]=$SCR_GRP[1].$MCH_POS_X;
:SR[24]=$SCR_GRP[1].$MCH_POS_Y;
3740: L P[3740] 800cm/min CNT100 COORD PTH ;
:SR[23]=$SCR_GRP[1].$MCH_POS_X;
:SR[24]=$SCR_GRP[1].$MCH_POS_Y;
3741: L P[3741] 800cm/min CNT100 COORD PTH ;
:SR[23]=$SCR_GRP[1].$MCH_POS_X;
:SR[24]=$SCR_GRP[1].$MCH_POS_Y;
3742: L P[3742] 800cm/min CNT100 COORD PTH ;
:SR[23]=$SCR_GRP[1].$MCH_POS_X;
:SR[24]=$SCR_GRP[1].$MCH_POS_Y;
3743: L P[3743] 800cm/min CNT100 COORD PTH ;
:SR[23]=$SCR_GRP[1].$MCH_POS_X;
:SR[24]=$SCR_GRP[1].$MCH_POS_Y;
3744: L P[3744] 800cm/min CNT100 COORD PTH ;
:SR[23]=$SCR_GRP[1].$MCH_POS_X;
:SR[24]=$SCR_GRP[1].$MCH_POS_Y;
3745: L P[3745] 800cm/min CNT100 COORD PTH ;
:SR[23]=$SCR_GRP[1].$MCH_POS_X;
:SR[24]=$SCR_GRP[1].$MCH_POS_Y;
3746: L P[3746] 800cm/min CNT100 COORD PTH ;
:SR[23]=$SCR_GRP[1].$MCH_POS_X;
:SR[24]=$SCR_GRP[1].$MCH_POS_Y;
3747: L P[3747] 800cm/min CNT100 COORD PTH ;
:SR[23]=$SCR_GRP[1].$MCH_POS_X;
:SR[24]=$SCR_GRP[1].$MCH_POS_Y;
3748: L P[3748] 800cm/min CNT100 COORD PTH ;
:SR[23]=$SCR_GRP[1].$MCH_POS_X;
:SR[24]=$SCR_GRP[1].$MCH_POS_Y;
3749: L P[3749] 800cm/min CNT100 COORD PTH ;
:SR[23]=$SCR_GRP[1].$MCH_POS_X;
:SR[24]=$SCR_GRP[1].$MCH_POS_Y;
3750: L P[3750] 800cm/min CNT100 COORD PTH ;
:SR[23]=$SCR_GRP[1].$MCH_POS_X;
:SR[24]=$SCR_GRP[1].$MCH_POS_Y;
3751: L P[3751] 800cm/min CNT100 COORD PTH ;
:SR[23]=$SCR_GRP[1].$MCH_POS_X;
:SR[24]=$SCR_GRP[1].$MCH_POS_Y;
3752: L P[3752] 800cm/min CNT100 COORD PTH ;
:SR[23]=$SCR_GRP[1].$MCH_POS_X;
:SR[24]=$SCR_GRP[1].$MCH_POS_Y;
3753: L P[3753] 800cm/min CNT100 COORD PTH ;
:SR[23]=$SCR_GRP[1].$MCH_POS_X;
:SR[24]=$SCR_GRP[1].$MCH_POS_Y;
3754: L P[3754] 800cm/min CNT100 COORD PTH ;
:SR[23]=$SCR_GRP[1].$MCH_POS_X;
:SR[24]=$SCR_GRP[1].$MCH_POS_Y;
3755: L P[3755] 800cm/min CNT100 COORD PTH ;
:SR[23]=$SCR_GRP[1].$MCH_POS_X;
:SR[24]=$SCR_GRP[1].$MCH_POS_Y;
3756: L P[3756] 800cm/min CNT100 COORD PTH ;
:SR[23]=$SCR_GRP[1].$MCH_POS_X;
:SR[24]=$SCR_GRP[1].$MCH_POS_Y;
3757: L P[3757] 800cm/min CNT100 COORD PTH ;
:SR[23]=$SCR_GRP[1].$MCH_POS_X;
:SR[24]=$SCR_GRP[1].$MCH_POS_Y;
3758: L P[3758] 800cm/min CNT100 COORD PTH ;
:SR[23]=$SCR_GRP[1].$MCH_POS_X;
:SR[24]=$SCR_GRP[1].$MCH_POS_Y;
3759: L P[3759] 800cm/min CNT100 COORD PTH ;
:SR[23]=$SCR_GRP[1].$MCH_POS_X;
:SR[24]=$SCR_GRP[1].$MCH_POS_Y;
3760: L P[3760] 800cm/min CNT100 COORD PTH ;
:SR[23]=$SCR_GRP[1].$MCH_POS_X;
:SR[24]=$SCR_GRP[1].$MCH_POS_Y;
3761: L P[3761] 800cm/min CNT100 COORD PTH ;
:SR[23]=$SCR_GRP[1].$MCH_POS_X;
:SR[24]=$SCR_GRP[1].$MCH_POS_Y;
3762: L P[3762] 800cm/min CNT100 COORD PTH ;
:SR[23]=$SCR_GRP[1].$MCH_POS_X;
:SR[24]=$SCR_GRP[1].$MCH_POS_Y;
3763: L P[3763] 800cm/min CNT100 COORD PTH ;
:SR[23]=$SCR_GRP[1].$MCH_POS_X;
:SR[24]=$SCR_GRP[1].$MCH_POS_Y;
3764: L P[3764] 800cm/min CNT100 COORD PTH ;
:SR[23]=$SCR_GRP[1].$MCH_POS_X;
:SR[24]=$SCR_GRP[1].$MCH_POS_Y;
3765: L P[3765] 800cm/min CNT100 COORD PTH ;
:SR[23]=$SCR_GRP[1].$MCH_POS_X;
:SR[24]=$SCR_GRP[1].$MCH_POS_Y;
3766: L P[3766] 800cm/min CNT100 COORD PTH ;
:SR[23]=$SCR_GRP[1].$MCH_POS_X;
:SR[24]=$SCR_GRP[1].$MCH_POS_Y;
3767: L P[3767] 800cm/min CNT100 COORD PTH ;
:SR[23]=$SCR_GRP[1].$MCH_POS_X;
:SR[24]=$SCR_GRP[1].$MCH_POS_Y;
3768: L P[3768] 800cm/min CNT100 COORD PTH ;
:SR[23]=$SCR_GRP[1].$MCH_POS_X;
:SR[24]=$SCR_GRP[1].$MCH_POS_Y;
3769: L P[3769] 800cm/min CNT100 COORD PTH ;
:SR[23]=$SCR_GRP[1].$MCH_POS_X;
:SR[24]=$SCR_GRP[1].$MCH_POS_Y;
3770: L P[3770] 800cm/min CNT100 COORD PTH ;
:SR[23]=$SCR_GRP[1].$MCH_POS_X;
:SR[24]=$SCR_GRP[1].$MCH_POS_Y;
3771: L P[3771] 800cm/min CNT100 COORD PTH ;
:SR[23]=$SCR_GRP[1].$MCH_POS_X;
:SR[24]=$SCR_GRP[1].$MCH_POS_Y;
3772: L P[3772] 800cm/min CNT100 COORD PTH ;
:SR[23]=$SCR_GRP[1].$MCH_POS_X;
:SR[24]=$SCR_GRP[1].$MCH_POS_Y;
3773: L P[3773] 800cm/min CNT100 COORD PTH ;
:SR[23]=$SCR_GRP[1].$MCH_POS_X;
:SR[24]=$SCR_GRP[1].$MCH_POS_Y;
3774: L P[3774] 800cm/min CNT100 COORD PTH ;
:SR[23]=$SCR_GRP[1].$MCH_POS_X;
:SR[24]=$SCR_GRP[1].$MCH_POS_Y;
3775: L P[3775] 800cm/min CNT100 COORD PTH ;
:SR[23]=$SCR_GRP[1].$MCH_POS_X;
:SR[24]=$SCR_GRP[1].$MCH_POS_Y;
3776: L P[3776] 800cm/min CNT100 COORD PTH ;
:SR[23]=$SCR_GRP[1].$MCH_POS_X;
:SR[24]=$SCR_GRP[1].$MCH_POS_Y;
3777: L P[3777] 800cm/min CNT100 COORD PTH ;
:SR[23]=$SCR_GRP[1].$MCH_POS_X;
:SR[24]=$SCR_GRP[1].$MCH_POS_Y;
3778: L P[3778] 800cm/min CNT100 COORD PTH ;
:SR[23]=$SCR_GRP[1].$MCH_POS_X;
:SR[24]=$SCR_GRP[1].$MCH_POS_Y;
3779: L P[3779] 800cm/min CNT100 COORD PTH ;
:SR[23]=$SCR_GRP[1].$MCH_POS_X;
:SR[24]=$SCR_GRP[1].$MCH_POS_Y;
3780: L P[3780] 800cm/min CNT100 COORD PTH ;
:SR[23]=$SCR_GRP[1].$MCH_POS_X;
:SR[24]=$SCR_GRP[1].$MCH_POS_Y;
3781: L P[3781] 800cm/min CNT100 COORD PTH ;
:SR[23]=$SCR_GRP[1].$MCH_POS_X;
:SR[24]=$SCR_GRP[1].$MCH_POS_Y;
3782: L P[3782] 800cm/min CNT100 COORD PTH ;
:SR[23]=$SCR_GRP[1].$MCH_POS_X;
:SR[24]=$SCR_GRP[1].$MCH_POS_Y;
3783: L P[3783] 800cm/min CNT100 COORD PTH ;
:SR[23]=$SCR_GRP[1].$MCH_POS_X;
:SR[24]=$SCR_GRP[1].$MCH_POS_Y;
3784: L P[3784] 800cm/min CNT100 COORD PTH ;
:SR[23]=$SCR_GRP[1].$MCH_POS_X;
:SR[24]=$SCR_GRP[1].$MCH_POS_Y;
3785: L P[3785] 800cm/min CNT100 COORD PTH ;
:SR[23]=$SCR_GRP[1].$MCH_POS_X;
:SR[24]=$SCR_GRP[1].$MCH_POS_Y;
3786: L P[3786] 800cm/min CNT100 COORD PTH ;
:SR[23]=$SCR_GRP[1].$MCH_POS_X;
:SR[24]=$SCR_GRP[1].$MCH_POS_Y;
3787: L P[3787] 800cm/min CNT100 COORD PTH ;
:SR[23]=$SCR_GRP[1].$MCH_POS_X;
:SR[24]=$SCR_GRP[1].$MCH_POS_Y;
3788: L P[3788] 800cm/min CNT100 COORD PTH ;
:SR[23]=$SCR_GRP[1].$MCH_POS_X;
:SR[24]=$SCR_GRP[1].$MCH_POS_Y;
3789: L P[3789] 800cm/min CNT100 COORD PTH ;
:SR[23]=$SCR_GRP[1].$MCH_POS_X;
:SR[24]=$SCR_GRP[1].$MCH_POS_Y;
3790: L P[3790] 800cm/min CNT100 COORD PTH ;
:SR[23]=$SCR_GRP[1].$MCH_POS_X;
:SR[24]=$SCR_GRP[1].$MCH_POS_Y;
3791: L P[3791] 800cm/min CNT100 COORD PTH ;
:SR[23]=$SCR_GRP[1].$MCH_POS_X;
:SR[24]=$SCR_GRP[1].$MCH_POS_Y;
3792: L P[3792] 800cm/min CNT100 COORD PTH ;
:SR[23]=$SCR_GRP[1].$MCH_POS_X;
:SR[24]=$SCR_GRP[1].$MCH_POS_Y;
3793: L P[3793] 800cm/min CNT100 COORD PTH ;
:SR[23]=$SCR_GRP[1].$MCH_POS_X;
:SR[24]=$SCR_GRP[1].$MCH_POS_Y;
3794: L P[3794] 800cm/min CNT100 COORD PTH ;
:SR[23]=$SCR_GRP[1].$MCH_POS_X;
:SR[24]=$SCR_GRP[1].$MCH_POS_Y;
3795: L P[3795] 800cm/min CNT100 COORD PTH ;
:SR[23]=$SCR_GRP[1].$MCH_POS_X;
:SR[24]=$SCR_GRP[1].$MCH_POS_Y;
3796: L P[3796] 800cm/min CNT100 COORD PTH ;
:SR[23]=$SCR_GRP[1].$MCH_POS_X;
:SR[24]=$SCR_GRP[1].$MCH_POS_Y;
3797: L P[3797] 800cm/min CNT100 COORD PTH ;
:SR[23]=$SCR_GRP[1].$MCH_POS_X;
:SR[24]=$SCR_GRP[1].$MCH_POS_Y;
3798: L P[3798] 800cm/min CNT100 COORD PTH ;
:SR[23]=$SCR_GRP[1].$MCH_POS_X;
:SR[24]=$SCR_GRP[1].$MCH_POS_Y;
3799: L P[3799] 800cm/min CNT100 COORD PTH ;
:SR[23]=$SCR_GRP[1].$MCH_POS_X;
:SR[24]=$SCR_GRP[1].$MCH_POS_Y;
3800: L P[3800] 800cm/min CNT100 COORD PTH ;
:SR[23]=$SCR_GRP[1].$MCH_POS_X;
:SR[24]=$SCR_GRP[1].$MCH_POS_Y;
3801: L P[3801] 800cm/min CNT100 COORD PTH ;
:SR[23]=$SCR_GRP[1].$MCH_POS_X;
:SR[24]=$SCR_GRP[1].$MCH_POS_Y;
3802: L P[3802] 800cm/min CNT100 COORD PTH ;
:SR[23]=$SCR_GRP[1].$MCH_POS_X;
:SR[24]=$SCR_GRP[1].$MCH_POS_Y;
3803: L P[3803] 800cm/min CNT100 COORD PTH ;
:SR[23]=$SCR_GRP[1].$MCH_POS_X;
:SR[24]=$SCR_GRP[1].$MCH_POS_Y;
3804: L P[3804] 800cm/min CNT100 COORD PTH ;
:SR[23]=$SCR_GRP[1].$MCH_POS_X;
:SR[24]=$SCR_GRP[1].$MCH_POS_Y;
3805: L P[3805] 800cm/min CNT100 COORD PTH ;
:SR[23]=$SCR_GRP[1].$MCH_POS_X;
:SR[24]=$SCR_GRP[1].$MCH_POS_Y;
3806: L P[3806] 800cm/min CNT100 COORD PTH ;
:SR[23]=$SCR_GRP[1].$MCH_POS_X;
:SR[24]=$SCR_GRP[1].$MCH_POS_Y;
3807: L P[3807] 800cm/min CNT100 COORD PTH ;
:SR[23]=$SCR_GRP[1].$MCH_POS_X;
:SR[24]=$SCR_GRP[1].$MCH_POS_Y;
3808: L P[3808] 800cm/min CNT100 COORD PTH ;
:SR[23]=$SCR_GRP[1].$MCH_POS_X;
:SR[24]=$SCR_GRP[1].$MCH_POS_Y;
3809: L P[3809] 800cm/min CNT100 COORD PTH ;
:SR[23]=$SCR_GRP[1].$MCH_POS_X;
:SR[24]=$SCR_GRP[1].$MCH_POS_Y;
3810: L P[3810] 800cm/min CNT100 COORD PTH ;
:SR[23]=$SCR_GRP[1].$MCH_POS_X;
:SR[24]=$SCR_GRP[1].$MCH_POS_Y;
3811: L P[3811] 800cm/min CNT100 COORD PTH ;
:SR[23]=$SCR_GRP[1].$MCH_POS_X;
:SR[24]=$SCR_GRP[1].$MCH_POS_Y;
3812: L P[3812] 800cm/min CNT100 COORD PTH ;
:SR[23]=$SCR_GRP[1].$MCH_POS_X;
:SR[24]=$SCR_GRP[1].$MCH_POS_Y;
3813: L P[3813] 800cm/min CNT100 COORD PTH ;
:SR[23]=$SCR_GRP[1].$MCH_POS_X;
:SR[24]=$SCR_GRP[1].$MCH_POS_Y;
3814: L P[3814] 800cm/min CNT100 COORD PTH ;
:SR[23]=$SCR_GRP[1].$MCH_POS_X;
:SR[24]=$SCR_GRP[1].$MCH_POS_Y;
3815: L P[3815] 800cm/min CNT100 COORD PTH ;
:SR[23]=$SCR_GRP[1].$MCH_POS_X;
:SR[24]=$SCR_GRP[1].$MCH_POS_Y;
3816: L P[3816] 800cm/min CNT100 COORD PTH ;
:SR[23]=$SCR_GRP[1].$MCH_POS_X;
:SR[24]=$SCR_GRP[1].$MCH_POS_Y;
3817: L P[3817] 800cm/min CNT100 COORD PTH ;
:SR[23]=$SCR_GRP[1].$MCH_POS_X;
:SR[24]=$SCR_GRP[1].$MCH_POS_Y;
3818: L P[3818] 800cm/min CNT100 COORD PTH ;
:SR[23]=$SCR_GRP[1].$MCH_POS_X;
:SR[24]=$SCR_GRP[1].$MCH_POS_Y;
3819: L P[3819] 800cm/min CNT100 COORD PTH ;
:SR[23]=$SCR_GRP[1].$MCH_POS_X;
:SR[24]=$SCR_GRP[1].$MCH_POS_Y;
3820: L P[3820] 800cm/min CNT100 COORD PTH ;
:SR[23]=$SCR_GRP[1].$MCH_POS_X;
:SR[24]=$SCR_GRP[1].$MCH_POS_Y;
3821: L P[3821] 800cm/min CNT100 COORD PTH ;
:SR[23]=$SCR_GRP[1].$MCH_POS_X;
:SR[24]=$SCR_GRP[1].$MCH_POS_Y;
3822: L P[3822] 800cm/min CNT100 COORD PTH ;
:SR[23]=$SCR_GRP[1].$MCH_POS_X;
:SR[24]=$SCR_GRP[1].$MCH_POS_Y;
3823: L P[3823] 800cm/min CNT100 COORD PTH ;
:SR[23]=$SCR_GRP[1].$MCH_POS_X;
:SR[24]=$SCR_GRP[1].$MCH_POS_Y;
3824: L P[3824] 800cm/min CNT100 COORD PTH ;
:SR[23]=$SCR_GRP[1].$MCH_POS_X;
:SR[24]=$SCR_GRP[1].$MCH_POS_Y;
3825: L P[3825] 800cm/min CNT100 COORD PTH ;
:SR[23]=$SCR_GRP[1].$MCH_POS_X;
:SR[24]=$SCR_GRP[1].$MCH_POS_Y;
3826: L P[3826] 800cm/min CNT100 COORD PTH ;
:SR[23]=$SCR_GRP[1].$MCH_POS_X;
:SR[24]=$SCR_GRP[1].$MCH_POS_Y;
3827: L P[3827] 800cm/min CNT100 COORD PTH ;
:SR[23]=$SCR_GRP[1].$MCH_POS_X;
:SR[24]=$SCR_GRP[1].$MCH_POS_Y;
3828: L P[3828] 800cm/min CNT100 COORD PTH ;
:SR[23]=$SCR_GRP[1].$MCH_POS_X;
:SR[24]=$SCR_GRP[1].$MCH_POS_Y;
3829: L P[3829] 800cm/min CNT100 COORD PTH ;
:SR[23]=$SCR_GRP[1].$MCH_POS_X;
:SR[24]=$SCR_GRP[1].$MCH_POS_Y;
3830: L P[3830] 800cm/min CNT100 COORD PTH ;
:SR[23]=$SCR_GRP[1].$MCH_POS_X;
:SR[24]=$SCR_GRP[1].$MCH_POS_Y;
3831: L P[3831] 800cm/min CNT100 COORD PTH ;
:SR[23]=$SCR_GRP[1].$MCH_POS_X;
:SR[24]=$SCR_GRP[1].$MCH_POS_Y;
3832: L P[3832] 800cm/min CNT100 COORD PTH ;
:SR[23]=$SCR_GRP[1].$MCH_POS_X;
:SR[24]=$SCR_GRP[1].$MCH_POS_Y;
3833: L P[3833] 800cm/min CNT100 COORD PTH ;
:SR[23]=$SCR_GRP[1].$MCH_POS_X;
:SR[24]=$SCR_GRP[1].$MCH_POS_Y;
3834: L P[3834] 800cm/min CNT100 COORD PTH ;
:SR[23]=$SCR_GRP[1].$MCH_POS_X;
:SR[24]=$SCR_GRP[1].$MCH_POS_Y;
3835: L P[3835] 800cm/min CNT100 COORD PTH ;
:SR[23]=$SCR_GRP[1].$MCH_POS_X;
:SR[24]=$SCR_GRP[1].$MCH_POS_Y;
3836: L P[3836] 800cm/min CNT100 COORD PTH ;
:SR[23]=$SCR_GRP[1].$MCH_POS_X;
:SR[24]=$SCR_GRP[1].$MCH_POS_Y;
3837: L P[3837] 800cm/min CNT100 COORD PTH ;
:SR[23]=$SCR_GRP[1].$MCH_POS_X;
:SR[24]=$SCR_GRP[1].$MCH_POS_Y;
3838: L P[3838] 800cm/min CNT100 COORD PTH ;
:SR[23]=$SCR_GRP[1].$MCH_POS_X;
:SR[24]=$SCR_GRP[1].$MCH_POS_Y;
3839: L P[3839] 800cm/min CNT100 COORD PTH ;
:SR[23]=$SCR_GRP[1].$MCH_POS_X;
:SR[24]=$SCR_GRP[1].$MCH_POS_Y;
3840: L P[3840] 800cm/min CNT100 COORD PTH ;
:SR[23]=$SCR_GRP[1].$MCH_POS_X;
:SR[24]=$SCR_GRP[1].$MCH_POS_Y;
3841: L P[3841] 800cm/min CNT100 COORD PTH ;
:SR[23]=$SCR_GRP[1].$MCH_POS_X;
:SR[24]=$SCR_GRP[1].$MCH_POS_Y;
3842: L P[3842] 800cm/min CNT100 COORD PTH ;
:SR[23]=$SCR_GRP[1].$MCH_POS_X;
:SR[24]=$SCR_GRP[1].$MCH_POS_Y;
3843: L P[3843] 800cm/min CNT100 COORD PTH ;
:SR[23]=$SCR_GRP[1].$MCH_POS_X;
:SR[24]=$SCR_GRP[1].$MCH_POS_Y;
3844: L P[3844] 800cm/min CNT100 COORD PTH ;
:SR[23]=$SCR_GRP[1].$MCH_POS_X;
:SR[24]=$SCR_GRP[1].$MCH_POS_Y;
3845: L P[3845] 800cm/min CNT100 COORD PTH ;
:SR[23]=$SCR_GRP[1].$MCH_POS_X;
:SR[24]=$SCR_GRP[1].$MCH_POS_Y;
3846: L P[3846] 800cm/min CNT100 COORD PTH ;
:SR[23]=$SCR_GRP[1].$MCH_POS_X;
:SR[24]=$SCR_GRP[1].$MCH_POS_Y;
3847: L P[3847] 800cm/min CNT100 COORD PTH ;
:SR[23]=$SCR_GRP[1].$MCH_POS_X;
:SR[24]=$SCR_GRP[1].$MCH_POS_Y;
3848: L P[3848] 800cm/min CNT100 COORD PTH ;
:SR[23]=$SCR_GRP[1].$MCH_POS_X;
:SR[24]=$SCR_GRP[1].$MCH_POS_Y;
3849: L P[3849] 800cm/min CNT100 COORD PTH ;
:SR[23]=$SCR_GRP[1].$MCH_POS_X;
:SR[24]=$SCR_GRP[1].$MCH_POS_Y;
3850: L P[3850] 800cm/min CNT100 COORD PTH ;
:SR[23]=$SCR_GRP[1].$MCH_POS_X;
:SR[24]=$SCR_GRP[1].$MCH_POS_Y;
3851: L P[3851] 800cm/min CNT100 COORD PTH ;
:SR[23]=$SCR_GRP[1].$MCH_POS_X;
:SR[24]=$SCR_GRP[1].$MCH_POS_Y;
3852: L P[3852] 800cm/min CNT100 COORD PTH ;
:SR[23]=$SCR_GRP[1].$MCH_POS_X;
:SR[24]=$SCR_GRP[1].$MCH_POS_Y;
3853: L P[3853] 800cm/min CNT100 COORD PTH ;
:SR[23]=$SCR_GRP[1].$MCH_POS_X;
:SR[24]=$SCR_GRP[1].$MCH_POS_Y;
3854: L P[3854] 800cm/min CNT100 COORD PTH ;
:SR[23]=$SCR_GRP[1].$MCH_POS_X;
:SR[24]=$SCR_GRP[1].$MCH_POS_Y;
3855: L P[3855] 800cm/min CNT100 COORD PTH ;
:SR[23]=$SCR_GRP[1].$MCH_POS_X;
:SR[24]=$SCR_GRP[1].$MCH_POS_Y;
3856: L P[3856] 800cm/min CNT100 COORD PTH ;
:SR[23]=$SCR_GRP[1].$MCH_POS_X;
:SR[24]=$SCR_GRP[1].$MCH_POS_Y;
3857: L P[3857] 800cm/min CNT100 COORD PTH ;
:SR[23]=$SCR_GRP[1].$MCH_POS_X;
:SR[24]=$SCR_GRP[1].$MCH_POS_Y;
3858: L P[3858] 800cm/min CNT100 COORD PTH ;
:SR[23]=$SCR_GRP[1].$MCH_POS_X;
:SR[24]=$SCR_GRP[1].$MCH_POS_Y;
3859: L P[3859] 800cm/min CNT100 COORD PTH ;
:SR[23]=$SCR_GRP[1].$MCH_POS_X;
:SR[24]=$SCR_GRP[1].$MCH_POS_Y;
3860: L P[3860] 800cm/min CNT100 COORD PTH ;
:SR[23]=$SCR_GRP[1].$MCH_POS_X;
:SR[24]=$SCR_GRP[1].$MCH_POS_Y;
3861: L P[3861] 800cm/min CNT100 COORD PTH ;
:SR[23]=$SCR_GRP[1].$MCH_POS_X;
:SR[24]=$SCR_GRP[1].$MCH_POS_Y;
3862: L P[3862] 800cm/min CNT100 COORD PTH ;
:SR[23]=$SCR_GRP[1].$MCH_POS_X;
:SR[24]=$SCR_GRP[1].$MCH_POS_Y;
3863: L P[3863] 800cm/min CNT100 COORD PTH ;
:SR[23]=$SCR_GRP[1].$MCH_POS_X;
:SR[24]=$SCR_GRP[1].$MCH_POS_Y;
3864: L P[3864] 800cm/min CNT100 COORD PTH ;
:SR[23]=$SCR_GRP[1].$MCH_POS_X;
:SR[24]=$SCR_GRP[1].$MCH_POS_Y;
3865: L P[3865] 800cm/min CNT100 COORD PTH ;
:SR[23]=$SCR_GRP[1].$MCH_POS_X;
:SR[24]=$SCR_GRP[1].$MCH_POS_Y;
3866: L P[3866] 800cm/min CNT100 COORD PTH ;
:SR[23]=$SCR_GRP[1].$MCH_POS_X;
:SR[24]=$SCR_GRP[1].$MCH_POS_Y;
3867: L P[3867] 800cm/min CNT100 COORD PTH ;
:SR[23]=$SCR_GRP[1].$MCH_POS_X;
:SR[24]=$SCR_GRP[1].$MCH_POS_Y;
3868: L P[3868] 800cm/min CNT100 COORD PTH ;
:SR[23]=$SCR_GRP[1].$MCH_POS_X;
:SR[24]=$SCR_GRP[1].$MCH_POS_Y;
3869: L P[3869] 800cm/min CNT100 COORD PTH ;
:SR[23]=$SCR_GRP[1].$MCH_POS_X;
:SR[24]=$SCR_GRP[1].$MCH_POS_Y;
3870: L P[3870] 800cm/min CNT100 COORD PTH ;
:SR[23]=$SCR_GRP[1].$MCH_POS_X;
:SR[24]=$SCR_GRP[1].$MCH_POS_Y;
3871: L P[3871] 800cm/min CNT100 COORD PTH ;
:SR[23]=$SCR_GRP[1].$MCH_POS_X;
:SR[24]=$SCR_GRP[1].$MCH_POS_Y;
3872: L P[3872] 800cm/min CNT100 COORD PTH ;
:SR[23]=$SCR_GRP[1].$MCH_POS_X;
:SR[24]=$SCR_GRP[1].$MCH_POS_Y;
3873: L P[3873] 800cm/min CNT100 COORD PTH ;
:SR[23]=$SCR_GRP[1].$MCH_POS_X;
:SR[24]=$SCR_GRP[1].$MCH_POS_Y;
3874: L P[3874] 800cm/min CNT100 COORD PTH ;
:SR[23]=$SCR_GRP[1].$MCH_POS_X;
:SR[24]=$SCR_GRP[1].$MCH_POS_Y;
3875: L P[3875] 800cm/min CNT100 COORD PTH ;
:SR[23]=$SCR_GRP[1].$MCH_POS_X;
:SR[24]=$SCR_GRP[1].$MCH_POS_Y;
3876: L P[3876] 800cm/min CNT100 COORD PTH ;
:SR[23]=$SCR_GRP[1].$MCH_POS_X;
:SR[24]=$SCR_GRP[1].$MCH_POS_Y;
3877: L P[3877] 800cm/min CNT100 COORD PTH ;
:SR[23]=$SCR_GRP[1].$MCH_POS_X;
:SR[24]=$SCR_GRP[1].$MCH_POS_Y;
3878: L P[3878] 800cm/min CNT100 COORD PTH ;
:SR[23]=$SCR_GRP[1].$MCH_POS_X;
:SR[24]=$SCR_GRP[1].$MCH_POS_Y;
3879: L P[3879] 800cm/min CNT100 COORD PTH ;
:SR[23]=$SCR_GRP[1].$MCH_POS_X;
:SR[24]=$SCR_GRP[1].$MCH_POS_Y;
3880: L P[3880] 800cm/min CNT100 COORD PTH ;
:SR[23]=$SCR_GRP[1].$MCH_POS_X;
:SR[24]=$SCR_GRP[1].$MCH_POS_Y;
3881: L P[3881] 800cm/min CNT100 COORD PTH ;
:SR[23]=$SCR_GRP[1].$MCH_POS_X;
:SR[24]=$SCR_GRP[1].$MCH_POS_Y;
3882: L P[3882] 800cm/min CNT100 COORD PTH ;
:SR[23]=$SCR_GRP[1].$MCH_POS_X;
:SR[24]=$SCR_GRP[1].$MCH_POS_Y;
3883: L P[3883] 800cm/min CNT100 COORD PTH ;
:SR[23]=$SCR_GRP[1].$MCH_POS_X;
:SR[24]=$SCR_GRP[1].$MCH_POS_Y;
3884: L P[3884] 800cm/min CNT100 COORD PTH ;
:SR[23]=$SCR_GRP[1].$MCH_POS_X;
:SR[24]=$SCR_GRP[1].$MCH_POS_Y;
3885: L P[3885] 800cm/min CNT100 COORD PTH ;
:SR[23]=$SCR_GRP[1].$MCH_POS_X;
:SR[24]=$SCR_GRP[1].$MCH_POS_Y;
3886: L P[3886] 800cm/min CNT100 COORD PTH ;
:SR[23]=$SCR_GRP[1].$MCH_POS_X;
:SR[24]=$SCR_GRP[1].$MCH_POS_Y;
3887: L P[3887] 800cm/min CNT100 COORD PTH ;
:SR[23]=$SCR_GRP[1].$MCH_POS_X;
:SR[24]=$SCR_GRP[1].$MCH_POS_Y;
3888: L P[3888] 800cm/min CNT100 COORD PTH ;
:SR[23]=$SCR_GRP[1].$MCH_POS_X;
:SR[24]=$SCR_GRP[1].$MCH_POS_Y;
3889: L P[3889] 800cm/min CNT100 COORD PTH ;
:SR[23]=$SCR_GRP[1].$MCH_POS_X;
:SR[24]=$SCR_GRP[1].$MCH_POS_Y;
3890: L P[3890] 800cm/min CNT100 COORD PTH ;
:SR[23]=$SCR_GRP[1].$MCH_POS_X;
:SR[24]=$SCR_GRP[1].$MCH_POS_Y;
3891: L P[3891] 800cm/min CNT100 COORD PTH ;
:SR[23]=$SCR_GRP[1].$MCH_POS_X;
:SR[24]=$SCR_GRP[1].$MCH_POS_Y;
3892: L P[3892] 800cm/min CNT100 COORD PTH ;
:SR[23]=$SCR_GRP[1].$MCH_POS_X;
:SR[24]=$SCR_GRP[1].$MCH_POS_Y;
3893: L P[3893] 800cm/min CNT100 COORD PTH ;
:SR[23]=$SCR_GRP[1].$MCH_POS_X;
:SR[24]=$SCR_GRP[1].$MCH_POS_Y;
3894: L P[3894] 800cm/min CNT100 COORD PTH ;
:SR[23]=$SCR_GRP[1].$MCH_POS_X;
:SR[24]=$SCR_GRP[1].$MCH_POS_Y;
3895: L P[3895] 800cm/min CNT100 COORD PTH ;
:SR[23]=$SCR_GRP[1].$MCH_POS_X;
:SR[24]=$SCR_GRP[1].$MCH_POS_Y;
3896: L P[3896] 800cm/min CNT100 COORD PTH ;
:SR[23]=$SCR_GRP[1].$MCH_POS_X;
:SR[24]=$SCR_GRP[1].$MCH_POS_Y;
3897: L P[3897] 800cm/min CNT100 COORD PTH ;
:SR[23]=$SCR_GRP[1].$MCH_POS_X;
:SR[24]=$SCR_GRP[1].$MCH_POS_Y;
3898: L P[3898] 800cm/min CNT100 COORD PTH ;
:SR[23]=$SCR_GRP[1].$MCH_POS_X;
:SR[24]=$SCR_GRP[1].$MCH_POS_Y;
3899: L P[3899] 800cm/min CNT100 COORD PTH ;
:SR[23]=$SCR_GRP[1].$MCH_POS_X;
:SR[24]=$SCR_GRP[1].$MCH_POS_Y;
3900: L P[3900] 800cm/min CNT100 COORD PTH ;
:SR[23]=$SCR_GRP[1].$MCH_POS_X;
:SR[24]=$SCR_GRP[1].$MCH_POS_Y;
3901: L P[3901] 800cm/min CNT100 COORD PTH ;
:SR[23]=$SCR_GRP[1].$MCH_POS_X;
:SR[24]=$SCR_GRP[1].$MCH_POS_Y;
3902: L P[3902] 800cm/min CNT100 COORD PTH ;
:SR[23]=$SCR_GRP[1].$MCH_POS_X;
:SR[24]=$SCR_GRP[1].$MCH_POS_Y;
3903: L P[3903] 800cm/min CNT100 COORD PTH ;
:SR[23]=$SCR_GRP[1].$MCH_POS_X;
:SR[24]=$SCR_GRP[1].$MCH_POS_Y;
3904: L P[3904] 800cm/min CNT100 COORD PTH ;
:SR[23]=$SCR_GRP[1].$MCH_POS_X;
:SR[24]=$SCR_GRP[1].$MCH_POS_Y;
3905: L P[3905] 800cm/min CNT100 COORD PTH ;
:SR[23]=$SCR_GRP[1].$MCH_POS_X;
:SR[24]=$SCR_GRP[1].$MCH_POS_Y;
3906: L P[3906] 800cm/min CNT100 COORD PTH ;
:SR[23]=$SCR_GRP[1].$MCH_POS_X;
:SR[24]=$SCR_GRP[1].$MCH_POS_Y;
3907: L P[3907] 800cm/min CNT100 COORD PTH ;
:SR[23]=$SCR_GRP[1].$MCH_POS_X;
:SR[24]=$SCR_GRP[1].$MCH_POS_Y;
3908: L P[3908] 800cm/min CNT100 COORD PTH ;
:SR[23]=$SCR_GRP[1].$MCH_POS_X;
:SR[24]=$SCR_GRP[1].$MCH_POS_Y;
3909: L P[3909] 800cm/min CNT100 COORD PTH ;
:SR[23]=$SCR_GRP[1].$MCH_POS_X;
:SR[24]=$SCR_GRP[1].$MCH_POS_Y;
3910: L P[3910] 800cm/min CNT100 COORD PTH ;
:SR[23]=$SCR_GRP[1].$MCH_POS_X;
:SR[24]=$SCR_GRP[1].$MCH_POS_Y;
3911: L P[3911] 800cm/min CNT100 COORD PTH ;
:SR[23]=$SCR_GRP[1].$MCH_POS_X;
:SR[24]=$SCR_GRP[1].$MCH_POS_Y;
3912: L P[3912] 800cm/min CNT100 COORD PTH ;
:SR[23]=$SCR_GRP[1].$MCH_POS_X;
:SR[24]=$SCR_GRP[1].$MCH_POS_Y;
3913: L P[3913] 800cm/min CNT100 COORD PTH ;
:SR[23]=$SCR_GRP[1].$MCH_POS_X;
:SR[24]=$SCR_GRP[1].$MCH_POS_Y;
3914: L P[3914] 800cm/min CNT100 COORD PTH ;
:SR[23]=$SCR_GRP[1].$MCH_POS_X;
:SR[24]=$SCR_GRP[1].$MCH_POS_Y;
3915: L P[3915] 800cm/min CNT100 COORD PTH ;
:SR[23]=$SCR_GRP[1].$MCH_POS_X;
:SR[24]=$SCR_GRP[1].$MCH_POS_Y;
3916: L P[3916] 800cm/min CNT100 COORD PTH ;
:SR[23]=$SCR_GRP[1].$MCH_POS_X;
:SR[24]=$SCR_GRP[1].$MCH_POS_Y;
3917: L P[3917] 800cm/min CNT100 COORD PTH ;
:SR[23]=$SCR_GRP[1].$MCH_POS_X;
:SR[24]=$SCR_GRP[1].$MCH_POS_Y;
3918: L P[3918] 800cm/min CNT100 COORD PTH ;
:SR[23]=$SCR_GRP[1].$MCH_POS_X;
:SR[24]=$SCR_GRP[1].$MCH_POS_Y;
3919: L P[3919] 800cm/min CNT100 COORD PTH ;
:SR[23]=$SCR_GRP[1].$MCH_POS_X;
:SR[24]=$SCR_GRP[1].$MCH_POS_Y;
3920: L P[3920] 800cm/min CNT100 COORD PTH ;
:SR[23]=$SCR_GRP[1].$MCH_POS_X;
:SR[24]=$SCR_GRP[1].$MCH_POS_Y;
3921: L P[3921] 800cm/min CNT100 COORD PTH ;
:SR[23]=$SCR_GRP[1].$MCH_POS_X;
:SR[24]=$SCR_GRP[1].$MCH_POS_Y;
3922: L P[3922] 800cm/min CNT100 COORD PTH ;
:SR[23]=$SCR_GRP[1].$MCH_POS_X;
:SR[24]=$SCR_GRP[1].$MCH_POS_Y;
3923: L P[3923] 800cm/min CNT100 COORD PTH ;
:SR[23]=$SCR_GRP[1].$MCH_POS_X;
:SR[24]=$SCR_GRP[1].$MCH_POS_Y;
3924: L P[3924] 800cm/min CNT100 COORD PTH ;
:SR[23]=$SCR_GRP[1].$MCH_POS_X;
:SR[24]=$SCR_GRP[1].$MCH_POS_Y;
3925: L P[3925] 800cm/min CNT100 COORD PTH ;
:SR[23]=$SCR_GRP[1].$MCH_POS_X;
:SR[24]=$SCR_GRP[1].$MCH_POS_Y;
3926: L P[3926] 800cm/min CNT100 COORD PTH ;
:SR[23]=$SCR_GRP[1].$MCH_POS_X;
:SR[24]=$SCR_GRP[1].$MCH_POS_Y;
3927: L P[3927] 800cm/min CNT100 COORD PTH ;
:SR[23]=$SCR_GRP[1].$MCH_POS_X;
:SR[24]=$SCR_GRP[1].$MCH_POS_Y;
3928: L P[3928] 800cm/min CNT100 COORD PTH ;
:SR[23]=$SCR_GRP[1].$MCH_POS_X;
:SR[24]=$SCR_GRP[1].$MCH_POS_Y;
3929: L P[3929] 800cm/min CNT100 COORD PTH ;
:SR[23]=$SCR_GRP[1].$MCH_POS_X;
:SR[24]=$SCR_GRP[1].$MCH_POS_Y;
3930: L P[3930] 800cm/min CNT100 COORD PTH ;
:SR[23]=$SCR_GRP[1].$MCH_POS_X;
:SR[24]=$SCR_GRP[1].$MCH_POS_Y;
3931: L P[3931] 800cm/min CNT100 COORD PTH ;
:SR[23]=$SCR_GRP[1].$MCH_POS_X;
:SR[24]=$SCR_GRP[1].$MCH_POS_Y;
3932: L P[3932] 800cm/min CNT100 COORD PTH ;
:SR[23]=$SCR_GRP[1].$MCH_POS_X;
:SR[24]=$SCR_GRP[1].$MCH_POS_Y;
3933: L P[3933] 800cm/min CNT100 COORD PTH ;
:SR[23]=$SCR_GRP[1].$MCH_POS_X;
:SR[24]=$SCR_GRP[1].$MCH_POS_Y;
3934: L P[3934] 800cm/min CNT100 COORD PTH ;
:SR[23]=$SCR_GRP[1].$MCH_POS_X;
:SR[24]=$SCR_GRP[1].$MCH_POS_Y;
3935: L P[3935] 800cm/min CNT100 COORD PTH ;
:SR[23]=$SCR_GRP[1].$MCH_POS_X;
:SR[24]=$SCR_GRP[1].$MCH_POS_Y;
3936: L P[3936] 800cm/min CNT100 COORD PTH ;
:SR[23]=$SCR_GRP[1].$MCH_POS_X;
:SR[24]=$SCR_GRP[1].$MCH_POS_Y;
3937: L P[3937] 800cm/min CNT100 COORD PTH ;
:SR[23]=$SCR_GRP[1].$MCH_POS_X;
:SR[24]=$SCR_GRP[1].$MCH_POS_Y;
3938: L P[3938] 800cm/min CNT100 COORD PTH ;
:SR[23]=$SCR_GRP[1].$MCH_POS_X;
:SR[24]=$SCR_GRP[1].$MCH_POS_Y;
3939: L P[3939] 800cm/min CNT100 COORD PTH ;
:SR[23]=$SCR_GRP[1].$MCH_POS_X;
:SR[24]=$SCR_GRP[1].$MCH_POS_Y;
3940: L P[3940] 800cm/min CNT100 COORD PTH ;
:SR[23]=$SCR_GRP[1].$MCH_POS_X;
:SR[24]=$SCR_GRP[1].$MCH_POS_Y;
3941: L P[3941] 800cm/min CNT100 COORD PTH ;
:SR[23]=$SCR_GRP[1].$MCH_POS_X;
:SR[24]=$SCR_GRP[1].$MCH_POS_Y;
3942: L P[3942] 800cm/min CNT100 COORD PTH ;
:SR[23]=$SCR_GRP[1].$MCH_POS_X;
:SR[24]=$SCR_GRP[1].$MCH_POS_Y;
3943: L P[3943] 800cm/min CNT100 COORD PTH ;
:SR[23]=$SCR_GRP[1].$MCH_POS_X;
:SR[24]=$SCR_GRP[1].$MCH_POS_Y;
3944: L P[3944] 800cm/min CNT100 COORD PTH ;
:SR[23]=$SCR_GRP[1].$MCH_POS_X;
:SR[24]=$SCR_GRP[1].$MCH_POS_Y;
3945: L P[3945] 800cm/min CNT100 COORD PTH ;
:SR[23]=$SCR_GRP[1].$MCH_POS_X;
:SR[24]=$SCR_GRP[1].$MCH_POS_Y;
3946: L P[3946] 800cm/min CNT100 COORD PTH ;
:SR[23]=$SCR_GRP[1].$MCH_POS_X;
:SR[24]=$SCR_GRP[1].$MCH_POS_Y;
3947: L P[3947] 800cm/min CNT100 COORD PTH ;
:SR[23]=$SCR_GRP[1].$MCH_POS_X;
:SR[24]=$SCR_GRP[1].$MCH_POS_Y;
3948: L P[3948] 800cm/min CNT100 COORD PTH ;
:SR[23]=$SCR_GRP[1].$MCH_POS_X;
:SR[24]=$SCR_GRP[1].$MCH_POS_Y;
3949: L P[3949] 800cm/min CNT100 COORD PTH ;
:SR[23]=$SCR_GRP[1].$MCH_POS_X;
:SR[24]=$SCR_GRP[1].$MCH_POS_Y;
3950: L P[3950] 800cm/min CNT100 COORD PTH ;
:SR[23]=$SCR_GRP[1].$MCH_POS_X;
:SR[24]=$SCR_GRP[1].$MCH_POS_Y;
3951: L P[3951] 800cm/min CNT100 COORD PTH ;
:SR[23]=$SCR_GRP[1].$MCH_POS_X;
:SR[24]=$SCR_GRP[1].$MCH_POS_Y;
3952: L P[3952] 800cm/min CNT100 COORD PTH ;
:SR[23]=$SCR_GRP[1].$MCH_POS_X;
:SR[24]=$SCR_GRP[1].$MCH_POS_Y;
3953: L P[3953] 800cm/min CNT100 COORD PTH ;
:SR[23]=$SCR_GRP[1].$MCH_POS_X;
:SR[24]=$SCR_GRP[1].$MCH_POS_Y;
3954: L P[3954] 800cm/min CNT100 COORD PTH ;
:SR[23]=$SCR_GRP[1].$MCH_POS_X;
:SR[24]=$SCR_GRP[1].$MCH_POS_Y;
3955: L P[3955] 800cm/min CNT100 COORD PTH ;
:SR[23]=$SCR_GRP[1].$MCH_POS_X;
:SR[24]=$SCR_GRP[1].$MCH_POS_Y;
3956: L P[3956] 800cm/min CNT100 COORD PTH ;
:SR[23]=$SCR_GRP[1].$MCH_POS_X;
:SR[24]=$SCR_GRP[1].$MCH_POS_Y;
3957: L P[3957] 800cm/min CNT100 COORD PTH ;
:SR[23]=$SCR_GRP[1].$MCH_POS_X;
:SR[24]=$SCR_GRP[1].$MCH_POS_Y;
3958: L P[3958] 800cm/min CNT100 COORD PTH ;
:SR[23]=$SCR_GRP[1].$MCH_POS_X;
:SR[24]=$SCR_GRP[1].$MCH_POS_Y;
3959: L P[3959] 800cm/min CNT100 COORD PTH ;
:SR[23]=$SCR_GRP[1].$MCH_POS_X;
:SR[24]=$SCR_GRP[1].$MCH_POS_Y;
3960: L P[3960] 800cm/min CNT100 COORD PTH ;
:SR[23]=$SCR_GRP[1].$MCH_POS_X;
:SR[24]=$SCR_GRP[1].$MCH_POS_Y;
3961: L P[3961] 800cm/min CNT100 COORD PTH ;
:SR[23]=$SCR_GRP[1].$MCH_POS_X;
:SR[24]=$SCR_GRP[1].$MCH_POS_Y;
3962: L P[3962] 800cm/min CNT100 COORD PTH ;
:SR[23]=$SCR_GRP[1].$MCH_POS_X;
:SR[24]=$SCR_GRP[1].$MCH_POS_Y;
3963: L P[3963] 800cm/min CNT100 COORD PTH ;
:SR[23]=$SCR_GRP[1].$MCH_POS_X;
:SR[24]=$SCR_GRP[1].$MCH_POS_Y;
3964: L P[3964] 800cm/min CNT100 COORD PTH ;
:SR[23]=$SCR_GRP[1].$MCH_POS_X;
:SR[24]=$SCR_GRP[1].$MCH_POS_Y;
3965: L P[3965] 800cm/min CNT100 COORD PTH ;
:SR[23]=$SCR_GRP[1].$MCH_POS_X;
:SR[24]=$SCR_GRP[1].$MCH_POS_Y;
3966: L P[3966] 800cm/min CNT100 COORD PTH ;
:SR[23]=$SCR_GRP[1].$MCH_POS_X;
:SR[24]=$SCR_GRP[1].$MCH_POS_Y;
3967: L P[3967] 800cm/min CNT100 COORD PTH ;
:SR[23]=$SCR_GRP[1].$MCH_POS_X;
:SR[24]=$SCR_GRP[1].$MCH_POS_Y;
3968: L P[3968] 800cm/min CNT100 COORD PTH ;
:SR[23]=$SCR_GRP[1].$MCH_POS_X;
:SR[24]=$SCR_GRP[1].$MCH_POS_Y;
3969: L P[3969] 800cm/min CNT100 COORD PTH ;
:SR[23]=$SCR_GRP[1].$MCH_POS_X;
:SR[24]=$SCR_GRP[1].$MCH_POS_Y;
3970: L P[3970] 800cm/min CNT100 COORD PTH ;
:SR[23]=$SCR_GRP[1].$MCH_POS_X;
:SR[24]=$SCR_GRP[1].$MCH_POS_Y;
3971: L P[3971] 800cm/min CNT100 COORD PTH ;
:SR[23]=$SCR_GRP[1].$MCH_POS_X;
:SR[24]=$SCR_GRP[1].$MCH_POS_Y;
3972: L P[3972] 800cm/min CNT100 COORD PTH ;
:SR[23]=$SCR_GRP[1].$MCH_POS_X;
:SR[24]=$SCR_GRP[1].$MCH_POS_Y;
3973: L P[3973] 800cm/min CNT100 COORD PTH ;
:SR[23]=$SCR_GRP[1].$MCH_POS_X;
:SR[24]=$SCR_GRP[1].$MCH_POS_Y;
3974: L P[3974] 800cm/min CNT100 COORD PTH ;
:SR[23]=$SCR_GRP[1].$MCH_POS_X;
:SR[24]=$SCR_GRP[1].$MCH_POS_Y;
3975: L P[3975] 800cm/min CNT100 COORD PTH ;
:SR[23]=$SCR_GRP[1].$MCH_POS_X;
:SR[24]=$SCR_GRP[1].$MCH_POS_Y;
3976: L P[3976] 800cm/min CNT100 COORD PTH ;
:SR[23]=$SCR_GRP[1].$MCH_POS_X;
:SR[24]=$SCR_GRP[1].$MCH_POS_Y;
3977: L P[3977] 800cm/min CNT100 COORD PTH ;
:SR[23]=$SCR_GRP[1].$MCH_POS_X;
:SR[24]=$SCR_GRP[1].$MCH_POS_Y;
3978: L P[3978] 800cm/min CNT100 COORD PTH ;
:SR[23]=$SCR_GRP[1].$MCH_POS_X;
:SR[24]=$SCR_GRP[1].$MCH_POS_Y;
3979: L P[3979] 800cm/min CNT100 COORD PTH ;
:SR[23]=$SCR_GRP[1].$MCH_POS_X;
:SR[24]=$SCR_GRP[1].$MCH_POS_Y;
3980: L P[3980] 800cm/min CNT100 COORD PTH ;
:SR[23]=$SCR_GRP[1].$MCH_POS_X;
:SR[24]=$SCR_GRP[1].$MCH_POS_Y;
3981: L P[3981] 800cm/min CNT100 COORD PTH ;
:SR[23]=$SCR_GRP[1].$MCH_POS_X;
:SR[24]=$SCR_GRP[1].$MCH_POS_Y;
3982: L P[3982] 800cm/min CNT100 COORD PTH ;
:SR[23]=$SCR_GRP[1].$MCH_POS_X;
:SR[24]=$SCR_GRP[1].$MCH_POS_Y;
3983: L P[3983] 800cm/min CNT100 COORD PTH ;
:SR[23]=$SCR_GRP[1].$MCH_POS_X;
:SR[24]=$SCR_GRP[1].$MCH_POS_Y;
3984: L P[3984] 800cm/min CNT100 COORD PTH ;
:SR[23]=$SCR_GRP[1].$MCH_POS_X;
:SR[24]=$SCR_GRP[1].$MCH_POS_Y;
3985: L P[3985] 800cm/min CNT100 COORD PTH ;
:SR[23]=$SCR_GRP[1].$MCH_POS_X;
:SR[24]=$SCR_GRP[1].$MCH_POS_Y;
3986: L P[3986] 800cm/min CNT100 COORD PTH ;
:SR[23]=$SCR_GRP[1].$MCH_POS_X;
:SR[24]=$SCR_GRP[1].$MCH_POS_Y;
3987: L P[3987] 800cm/min CNT100 COORD PTH ;
:SR[23]=$SCR_GRP[1].$MCH_POS_X;
:SR[24]=$SCR_GRP[1].$MCH_POS_Y;
3988: L P[3988] 800cm/min CNT100 COORD PTH ;
:SR[23]=$SCR_GRP[1].$MCH_POS_X;
:SR[24]=$SCR_GRP[1].$MCH_POS_Y;
3989: L P[3989] 800cm/min CNT100 COORD PTH ;
:SR[23]=$SCR_GRP[1].$MCH_POS_X;
:SR[24]=$SCR_GRP[1].$MCH_POS_Y;
3990: L P[3990] 800cm/min CNT100 COORD PTH ;
:SR[23]=$SCR_GRP[1].$MCH_POS_X;
:SR[24]=$SCR_GRP[1].$MCH_POS_Y;
3991: L P[3991] 800cm/min CNT100 COORD PTH ;
:SR[23]=$SCR_GRP[1].$MCH_POS_X;
:SR[24]=$SCR_GRP[1].$MCH_POS_Y;
3992: L P[3992] 800cm/min CNT100 COORD PTH ;
:SR[23]=$SCR_GRP[1].$MCH_POS_X;
:SR[24]=$SCR_GRP[1].$MCH_POS_Y;
3993: L P[3993] 800cm/min CNT100 COORD PTH ;
:SR[23]=$SCR_GRP[1].$MCH_POS_X;
:SR[24]=$SCR_GRP[1].$MCH_POS_Y;
3994: L P[3994] 800cm/min CNT100 COORD PTH ;
:SR[23]=$SCR_GRP[1].$MCH_POS_X;
:SR[24]=$SCR_GRP[1].$MCH_POS_Y;
3995: L P[3995] 800cm/min CNT100 COORD PTH ;
:SR[23]=$SCR_GRP[1].$MCH_POS_X;
:SR[24]=$SCR_GRP[1].$MCH_POS_Y;
3996: L P[3996] 800cm/min CNT100 COORD PTH ;
:SR[23]=$SCR_GRP[1].$MCH_POS_X;
:SR[24]=$SCR_GRP[1].$MCH_POS_Y;
3997: L P[3997] 800cm/min CNT100 COORD PTH ;
:SR[23]=$SCR_GRP[1].$MCH_POS_X;
:SR[24]=$SCR_GRP[1].$MCH_POS_Y;
3998: L P[3998] 800cm/min CNT100 COORD PTH ;
:SR[23]=$SCR_GRP[1].$MCH_POS_X;
:SR[24]=$SCR_GRP[1].$MCH_POS_Y;
3999: L P[3999] 800cm/min CNT100 COORD PTH ;
:SR[23]=$SCR_GRP[1].$MCH_POS_X;
:SR[24]=$SCR_GRP[1].$MCH_POS_Y;
4000: L P[4000] 800cm/min CNT100 COORD PTH ;
:SR[23]=$SCR_GRP[1].$MCH_POS_X;
:SR[24]=$SCR_GRP[1].$MCH_POS_Y;
4001: L P[4001] 800cm/min CNT100 COORD PTH ;
:SR[23]=$SCR_GRP[1].$MCH_POS_X;
:SR[24]=$SCR_GRP[1].$MCH_POS_Y;
4002: L P[4002] 800cm/min CNT100 COORD PTH ;
:SR[23]=$SCR_GRP[1].$MCH_POS_X;
:SR[24]=$SCR_GRP[1].$MCH_POS_Y;
4003: L P[4003] 800cm/min CNT100 COORD PTH ;
:SR[23]=$SCR_GRP[1].$MCH_POS_X;
:SR[24]=$SCR_GRP[1].$MCH_POS_Y;
4004: L P[4004] 800cm/min CNT100 COORD PTH ;
:SR[23]=$SCR_GRP[1].$MCH_POS_X;
:SR[24]=$SCR_GRP[1].$MCH_POS_Y;
4005: L P[4005] 800cm/min CNT100 COORD PTH ;
:SR[23]=$SCR_GRP[1].$MCH_POS_X;
:SR[24]=$SCR_GRP[1].$MCH_POS_Y;
4006: L P[4006] 800cm/min CNT100 COORD PTH ;
:SR[23]=$SCR_GRP[1].$MCH_POS_X;
:SR[24]=$SCR_GRP[1].$MCH_POS_Y;
4007: L P[4007] 800cm/min CNT100 COORD PTH ;
:SR[23]=$SCR_GRP[1].$MCH_POS_X;
:SR[24]=$SCR_GRP[1].$MCH_POS_Y;
4008: L P[4008] 800cm/min CNT100 COORD PTH ;
:SR[23]=$SCR_GRP[1].$MCH_POS_X;
:SR[24]=$SCR_GRP[1].$MCH_POS_Y;
4009: L P[4009] 800cm/min CNT100 COORD PTH ;
:SR[23]=$SCR_GRP[1].$MCH_POS_X;
:SR[24]=$SCR_GRP[1].$MCH_POS_Y;
4010: L P[4010] 800cm/min CNT100 COORD PTH ;
:SR[23]=$SCR_GRP[1].$MCH_POS_X;
:SR[24]=$SCR_GRP[1].$MCH_POS_Y;
4011: L P[4011] 800cm/min CNT100 COORD PTH ;
:SR[23]=$SCR_GRP[1].$MCH_POS_X;
:SR[24]=$SCR_GRP[1].$MCH_POS_Y;
4012: L P[4012] 800cm/min CNT100 COORD PTH ;
:SR[23]=$SCR_GRP[1].$MCH_POS_X;
:SR[24]=$SCR_GRP[1].$MCH_POS_Y;
4013: L P[4013] 800cm/min CNT100 COORD PTH ;
:SR[23]=$SCR_GRP[1].$MCH_POS_X;
:SR[24]=$SCR_GRP[1].$MCH_POS_Y;
4014: L P[4014] 800cm/min CNT100 COORD PTH ;
:SR[23]=$SCR_GRP[1].$MCH_POS_X;
:SR[24]=$SCR_GRP[1].$MCH_POS_Y;
4015: L P[4015] 800cm/min CNT100 COORD PTH ;
:SR[23]=$SCR_GRP[1].$MCH_POS_X;
:SR[24]=$SCR_GRP[1].$MCH_POS_Y;
4016: L P[4016] 800cm/min CNT100 COORD PTH ;
:SR[23]=$SCR_GRP[1].$MCH_POS_X;
:SR[24]=$SCR_GRP[1].$MCH_POS_Y;
4017: L P[4017] 800cm/min CNT100 COORD PTH ;
:SR[23]=$SCR_GRP[1].$MCH_POS_X;
:SR[24]=$SCR_GRP[1].$MCH_POS_Y;
4018: L P[4018] 800cm/min CNT100 COORD PTH ;
:SR[23]=$SCR_GRP[1].$MCH_POS_X;
:SR[24]=$SCR_GRP[1].$MCH_POS_Y;
4019: L P[4019] 800cm/min CNT100 COORD PTH ;
:SR[23]=$SCR_GRP[1].$MCH_POS_X;
:SR[24]=$SCR_GRP[1].$MCH_POS_Y;
4020: L P[4020] 800cm/min CNT100 COORD PTH ;
:SR[23]=$SCR_GRP[1].$MCH_POS_X;
:SR[24]=$SCR_GRP[1].$MCH_POS_Y;
4021: L P[4021] 800cm/min CNT100 COORD PTH ;
:SR[23]=$SCR_GRP[1].$MCH_POS_X;
:SR[24]=$SCR_GRP[1].$MCH_POS_Y;
4022: L P[4022] 800cm/min CNT100 COORD PTH ;
:SR[23]=$SCR_GRP[1].$MCH_POS_X;
:SR[24]=$SCR_GRP[1].$MCH_POS_Y;
4023: L P[4023] 800cm/min CNT100 COORD PTH ;
:SR[23]=$SCR_GRP[1].$MCH_POS_X;
:SR[24]=$SCR_GRP[1].$MCH_POS_Y;
4024: L P[4024] 800cm/min CNT100 COORD PTH ;
:SR[23]=$SCR_GRP[1].$MCH_POS_X;
:SR[24]=$SCR_GRP[1].$MCH_POS_Y;
4025: L P[4025] 800cm/min CNT100 COORD PTH ;
:SR[23]=$SCR_GRP[1].$MCH_POS_X;
:SR[24]=$SCR_GRP[1].$MCH_POS_Y;
4026: L P[4026] 800cm/min CNT100 COORD PTH ;
:SR[23]=$SCR_GRP[1].$MCH_POS_X;
:SR[24]=$SCR_GRP[1].$MCH_POS_Y;
4027: L P[4027] 800cm/min CNT100 COORD PTH ;
:SR[23]=$SCR_GRP[1].$MCH_POS_X;
:SR[24]=$SCR_GRP[1].$MCH_POS_Y;
4028: L P[4028] 800cm/min CNT100 COORD PTH ;
:SR[23]=$SCR_GRP[1].$MCH_POS_X;
:SR[24]=$SCR_GRP[1].$MCH_POS_Y;
4029: L P[4029] 800cm/min CNT100 COORD PTH ;
:SR[23]=$SCR_GRP[1].$MCH_POS_X;
:SR[24]=$SCR_GRP[1].$MCH_POS_Y;
4030: L P[4030] 800cm/min CNT100 COORD PTH ;
:SR[23]=$SCR_GRP[1].$MCH_POS_X;
:SR[24]=$SCR_GRP[1].$MCH_POS_Y;
4031: L P[4031] 800cm/min CNT100 COORD PTH ;
:SR[23]=$SCR_GRP[1].$MCH_POS_X;
:SR[24]=$SCR_GRP[1].$MCH_POS_Y;
4032: L P[4032] 800cm/min CNT100 COORD PTH ;
:SR[23]=$SCR_GRP[1].$MCH_POS_X;
:SR[24]=$SCR_GRP[1].$MCH_POS_Y;
4033: L P[4033] 800cm/min CNT100 COORD PTH ;
:SR[23]=$SCR_GRP[1].$MCH_POS_X;
:SR[24]=$SCR_GRP[1].$MCH_POS_Y;
4034: L P[4034] 800cm/min CNT100 COORD PTH ;
:SR[23]=$SCR_GRP[1].$MCH_POS_X;
:SR[24]=$SCR_GRP[1].$MCH_POS_Y;
4035: L P[4035] 800cm/min CNT100 COORD PTH ;
:SR[23]=$SCR_GRP[1].$MCH_POS_X;
:SR[24]=$SCR_GRP[1].$MCH_POS_Y;
4036: L P[4036] 800cm/min CNT100 COORD PTH ;
:SR[23]=$SCR_GRP[1].$MCH_POS_X;
:SR[24]=$SCR_GRP[1].$MCH_POS_Y;
4037: L P[4037] 800cm/min CNT100 COORD PTH ;
:SR[23]=$SCR_GRP[1].$MCH_POS_X;
:SR[24]=$SCR_GRP[1].$MCH_POS_Y;
4038: L P[4038] 800cm/min CNT100 COORD PTH ;
:SR[23]=$SCR_GRP[1].$MCH_POS_X;
:SR[24]=$SCR_GRP[1].$MCH_POS_Y;
4039: L P[4039] 800cm/min CNT100 COORD PTH ;
:SR[23]=$SCR_GRP[1].$MCH_POS_X;
:SR[24]=$SCR_GRP[1].$MCH_POS_Y;
4040: L P[4040] 800cm/min CNT100 COORD PTH ;
:SR[23]=$SCR_GRP[1].$MCH_POS_X;
:SR[24]=$SCR_GRP[1].$MCH_POS_Y;
4041: L P[4041] 800cm/min CNT100 COORD PTH ;
:SR[23]=$SCR_GRP[1].$MCH_POS_X;
:SR[24]=$SCR_GRP[1].$MCH_POS_Y;
4042: L P[4042] 800cm/min CNT100 COORD PTH ;
:SR[23]=$SCR_GRP[1].$MCH_POS_X;
:SR[24]=$SCR_GRP[1].$MCH_POS_Y;
4043: L P[4043] 800cm/min CNT100 COORD PTH ;
:SR[23]=$SCR_GRP[1].$MCH_POS_X;
:SR[24]=$SCR_GRP[1].$MCH_POS_Y;
4044: L P[4044] 800cm/min CNT100 COORD PTH ;
:SR[23]=$SCR_GRP[1].$MCH_POS_X;
:SR[24]=$SCR_GRP[1].$MCH_POS_Y;
4045: L P[4045] 800cm/min CNT100 COORD PTH ;
:SR[23]=$SCR_GRP[1].$MCH_POS_X;
:SR[24]=$SCR_GRP[1].$MCH_POS_Y;
4046: L P[4046] 800cm/min CNT100 COORD PTH ;
:SR[23]=$SCR_GRP[1].$MCH_POS_X;
:SR[24]=$SCR_GRP[1].$MCH_POS_Y;
4047: L P[4047] 800cm/min CNT100 COORD PTH ;
:SR[23]=$SCR_GRP[1].$MCH_POS_X;
:SR[24]=$SCR_GRP[1].$MCH_POS_Y;
4048: L P[4048] 800cm/min CNT100 COORD PTH ;
:SR[23]=$SCR_GRP[1].$MCH_POS_X;
:SR[24]=$SCR_GRP[1].$MCH_POS_Y;
4049: L P[4049] 800cm/min CNT100 COORD PTH ;
:SR[23]=$SCR_GRP[1].$MCH_POS_X;
:SR[24]=$SCR_GRP[1].$MCH_POS_Y;
4050: L P[4050] 800cm/min CNT100 COORD PTH ;
:SR[23]=$SCR_GRP[1].$MCH_POS_X;
:SR[24]=$SCR_GRP[1].$MCH_POS_Y;
4051: L P[4051] 800cm/min CNT100 COORD PTH ;
:SR[23]=$SCR_GRP[1].$MCH_POS_X;
:SR[24]=$SCR_GRP[1].$MCH_POS_Y;
4052: L P[4052] 800cm/min CNT100 COORD PTH ;
:SR[23]=$SCR_GRP[1].$MCH_POS_X;
:SR[24]=$SCR_GRP[1].$MCH_POS_Y;
4053: L P[4053] 800cm/min CNT100 COORD PTH ;
:SR[23]=$SCR_GRP[1].$MCH_POS_X;
:SR[24]=$SCR_GRP[1].$MCH_POS_Y;
4054: L P[4054] 800cm/min CNT100 COORD PTH ;
:SR[23]=$SCR_GRP[1].$MCH_POS_X;
:SR[24]=$SCR_GRP[1].$MCH_POS_Y;
4055: L P[4055] 800cm/min CNT100 COORD PTH ;
:SR[23]=$SCR_GRP[1].$MCH_POS_X;
:SR[24]=$SCR_GRP[1].$MCH_POS_Y;
4056: L P[4056] 800cm/min CNT100 COORD PTH ;
:SR[23]=$SCR_GRP[1].$MCH_POS_X;
:SR[24]=$SCR_GRP[1].$MCH_POS_Y;
4057: L P[4057] 800cm/min CNT100 COORD PTH ;
:SR[23]=$SCR_GRP[1].$MCH_POS_X;
:SR[24]=$SCR_GRP[1].$MCH_POS_Y;
4058: L P[4058] 800cm/min CNT100 COORD PTH ;
:SR[23]=$SCR_GRP[1].$MCH_POS_X;
:SR[24]=$SCR_GRP[1].$MCH_POS_Y;
4059: L P[4059] 800cm/min CNT100 COORD PTH ;
:SR[23]=$SCR_GRP[1].$MCH_POS_X;
:SR[24]=$SCR_GRP[1].$MCH_POS_Y;
4060: L P[4060] 800cm/min CNT100 COORD PTH ;
:SR[23]=$SCR_GRP[1].$MCH_POS_X;
:SR[24]=$SCR_GRP[1].$MCH_POS_Y;
4061: L P[4061] 800cm/min CNT100 COORD PTH ;
:SR[23]=$SCR_GRP[1].$MCH_POS_X;
:SR[24]=$SCR_GRP[1].$MCH_POS_Y;
4062: L P[4062] 800cm/min CNT100 COORD PTH ;
:SR[23]=$SCR_GRP[1].$MCH_POS_X;
:SR[24]=$SCR_GRP[1].$MCH_POS_Y;
4063: L P[4063] 800cm/min CNT100 COORD PTH ;
:SR[23]=$SCR_GRP[1].$MCH_POS_X;
:SR[24]=$SCR_GRP[1].$MCH_POS_Y;
4064: L P[4064] 800cm/min CNT100 COORD PTH ;
:SR[23]=$SCR_GRP[1].$MCH_POS_X;
:SR[24]=$SCR_GRP[1].$MCH_POS_Y;
4065: L P[4065] 800cm/min CNT100 COORD PTH ;
:SR[23]=$SCR_GRP[1].$MCH_POS_X;
:SR[24]=$SCR_GRP[1].$MCH_POS_Y;
4066: L P[4066] 800cm/min CNT100 COORD PTH ;
:SR[23]=$SCR_GRP[1].$MCH_POS_X;
:SR[24]=$SCR_GRP[1].$MCH_POS_Y;
4067: L P[4067] 800cm/min CNT100 COORD PTH ;
:SR[23]=$SCR_GRP[1].$MCH_POS_X;
:SR[24]=$SCR_GRP[1].$MCH_POS_Y;
4068: L P[4068] 800cm/min CNT100 COORD PTH ;
:SR[23]=$SCR_GRP[1].$MCH_POS_X;
:SR[24]=$SCR_GRP[1].$MCH_POS_Y;
4069: L P[4069] 800cm/min CNT100 COORD PTH ;
:SR[23]=$SCR_GRP[1].$MCH_POS_X;
:SR[24]=$SCR_GRP[1].$MCH_POS_Y;
4070: L P[4070] 800cm/min CNT100 COORD PTH ;
:SR[23]=$SCR_GRP[1].$MCH_POS_X;
:SR[24]=$SCR_GRP[1].$MCH_POS_Y;
4071: L P[4071] 800cm/min CNT100 COORD PTH ;
:SR[23]=$SCR_GRP[1].$MCH_POS_X;
:SR[24]=$SCR_GRP[1].$MCH_POS_Y;
4072: L P[4072] 800cm/min CNT100 COORD PTH ;
:SR[23]=$SCR_GRP[1].$MCH_POS_X;
:SR[24]=$SCR_GRP[1].$MCH_POS_Y;
4073: L P[4073] 800cm/min CNT100 COORD PTH ;
:SR[23]=$SCR_GRP[1].$MCH_POS_X;
:SR[24]=$SCR_GRP[1].$MCH_POS_Y;
4074: L P[4074] 800cm/min CNT100 COORD PTH ;
:SR[23]=$SCR_GRP[1].$MCH_POS_X;
:SR[24]=$SCR_GRP[1].$MCH_POS_Y;
4075: L P[4075] 800cm/min CNT100 COORD PTH ;
:SR[23]=$SCR_GRP[1].$MCH_POS_X;
:SR[24]=$SCR_GRP[1].$MCH_POS_Y;
4076: L P[4076] 800cm/min CNT100 COORD PTH ;
:SR[23]=$SCR_GRP[1].$MCH_POS_X;
:SR[24]=$SCR_GRP[1].$MCH_POS_Y;
4077: L P[4077] 800cm/min CNT100 COORD PTH ;
:SR[23]=$SCR_GRP[1].$MCH_POS_X;
:SR[24]=$SCR_GRP[1].$MCH_POS_Y;
4078: L P[4078] 800cm/min CNT100 COORD PTH ;
:SR[23]=$SCR_GRP[1].$MCH_POS_X;
:SR[24]=$SCR_GRP[1].$MCH_POS_Y;
4079: L P[4079] 800cm/min CNT100 COORD PTH ;
:SR[23]=$SCR_GRP[1].$MCH_POS_X;
:SR[24]=$SCR_GRP[1].$MCH_POS_Y;
4080: L P[4080] 800cm/min CNT100 COORD PTH ;
:SR[23]=$SCR_GRP[1].$MCH_POS_X;
:SR[24]=$SCR_GRP[1].$MCH_POS_Y;
4081: L P[4081] 800cm/min CNT100 COORD PTH ;
:SR[23]=$SCR_GRP[1].$MCH_POS_X;
:SR[24]=$SCR_GRP[1].$MCH_POS_Y;
4082: L P[4082] 800cm/min CNT100 COORD PTH ;
:SR[23]=$SCR_GRP[1].$MCH_POS_X;
:SR[24]=$SCR_GRP[1].$MCH_POS_Y;
4083: L P[4083] 800cm/min CNT100 COORD PTH ;
:SR[23]=$SCR_GRP[1].$MCH_POS_X;
:SR[24]=$SCR_GRP[1].$MCH_POS_Y;
4084: L P[4084] 800cm/min CNT100 COORD PTH ;
:SR[23]=$SCR_GRP[1].$MCH_POS_X;
:SR[24]=$SCR_GRP[1].$MCH_POS_Y;
4085: L P[4085] 800cm/min CNT100 COORD PTH ;
:SR[23]=$SCR_GRP[1].$MCH_POS_X;
:SR[24]=$SCR_GRP[1].$MCH_POS_Y;
4086: L P[4086] 800cm/min CNT100 COORD PTH ;
:SR[23]=$SCR_GRP[1].$MCH_POS_X;
:SR[24]=$SCR_GRP[1].$MCH_POS_Y;
4087: L P[4087] 800cm/min CNT100 COORD PTH ;
:SR[23]=$SCR_GRP[1].$MCH_POS_X;
:SR[24]=$SCR_GRP[1].$MCH_POS_Y;
4088: L P[4088] 800cm/min CNT100 COORD PTH ;
:SR[23]=$SCR_GRP[1].$MCH_POS_X;
:SR[24]=$SCR_GRP[1].$MCH_POS_Y;
4089: L P[4089] 800cm/min CNT100 COORD PTH ;
:SR[23]=$SCR_GRP[1].$MCH_POS_X;
:SR[24]=$SCR_GRP[1].$MCH_POS_Y;
4090: L P[4090] 800cm/min CNT100 COORD PTH ;
:SR[23]=$SCR_GRP[1].$MCH_POS_X;
:SR[24]=$SCR_GRP[1].$MCH_POS_Y;
4091: L P[4091] 800cm/min CNT100 COORD PTH ;
:SR[23]=$SCR_GRP[1].$MCH_POS_X;
:SR[24]=$SCR_GRP[1].$MCH_POS_Y;
4092: L P[4092] 800cm/min CNT100 COORD PTH ;
:SR[23]=$SCR_GRP[1].$MCH_POS_X;
:SR[24]=$SCR_GRP[1].$MCH_POS_Y;
4093: L P[4093] 800cm/min CNT100 COORD PTH ;
:SR[23]=$SCR_GRP[1].$MCH_POS_X;
:SR[24]=$SCR_GRP[1].$MCH_POS_Y;
4094: L P[4094] 800cm/min CNT100 COORD PTH ;
:SR[23]=$SCR_GRP[1].$MCH_POS_X;
:SR[24]=$SCR_GRP[1].$MCH_POS_Y;
4095: L P[4095] 800cm/min CNT100 COORD PTH ;
:SR[23]=$SCR_GRP[1].$MCH_POS_X;
:SR[24]=$SCR_GRP[1].$MCH_POS_Y;
4096: L P[4096] 800cm/min CNT100 COORD PTH ;
:SR[23]=$SCR_GRP[1].$MCH_POS_X;
:SR[24]=$SCR_GRP[1].$MCH_POS_Y;
4097: L P[4097] 800cm/min CNT100 COORD PTH ;
:SR[23]=$SCR_GRP[1].$MCH_POS_X;
:SR[24]=$SCR_GRP[1].$MCH_POS_Y;
4098: L P[4098] 800cm/min CNT100 COORD PTH ;
:SR[23]=$SCR_GRP[1].$MCH_POS_X;
:SR[24]=$SCR_GRP[1].$MCH_POS_Y;
4099: L P[4099] 800cm/min CNT100 COORD PTH ;
:SR[23]=$SCR_GRP[1].$MCH_POS_X;
:SR[24]=$SCR_GRP[1].$MCH_POS_Y;
4100: L P[4100] 800cm/min CNT100 COORD PTH ;
:SR[23]=$SCR_GRP[1].$MCH_POS_X;
:SR[24]=$SCR_GRP[1].$MCH_POS_Y;
4101: L P[4101] 800cm/min CNT100 COORD PTH ;
:SR[23]=$SCR_GRP[1].$MCH_POS_X;
:SR[24]=$SCR_GRP[1].$MCH_POS_Y;
4102: L P[4102] 800cm/min CNT100 COORD PTH ;
:SR[23]=$SCR_GRP[1].$MCH_POS_X;
:SR[24]=$SCR_GRP[1].$MCH_POS_Y;
4103: L P[4103] 800cm/min CNT100 COORD PTH ;
:SR[23]=$SCR_GRP[1].$MCH_POS_X;
:SR[24]=$SCR_GRP[1].$MCH_POS_Y;
4104: L P[4104] 800cm/min CNT100 COORD PTH ;
